Yaskawa INFORM job: DEMO_ROOF_UPPER_0625_3PAINT_39.JBI

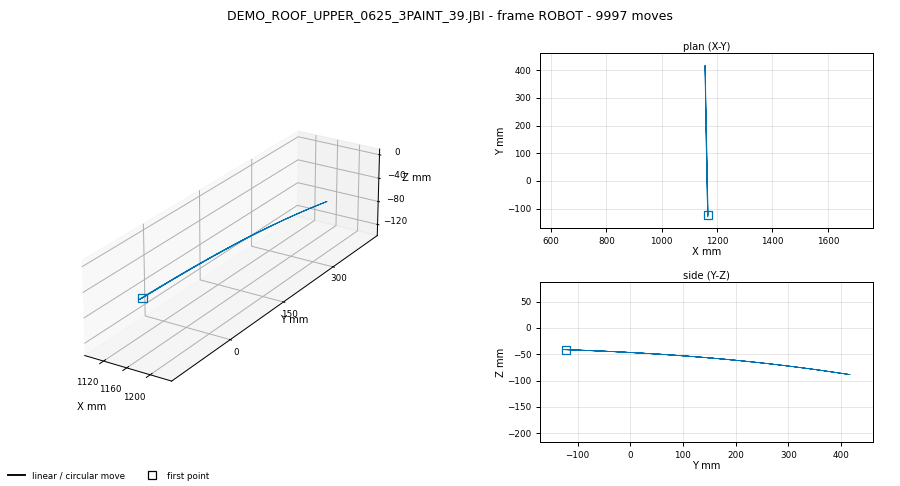
[picture p0: tool path of DEMO_ROOF_UPPER_0625_3PAINT_39.JBI in frame ROBOT, 9997 of 9997 moves have a stored position in this frame; points joined in program order, loops and branches not executed]
/JOB
//NAME DEMO_ROOF_UPPER_0625_3PAINT39
//POS
///NPOS 9997,0,0,0,0,0
///TOOL 0
///USER 0
///POSTYPE ROBOT
///RECTAN
///RCONF 1,0,0,0,0,0,0,0,0,0,0,0,0,0,0,0,0,0,0,0,0,0,0,0
C00000=1167.376,-121.731,-41.179,178.758,5.790,149.399
C00001=1167.371,-121.482,-41.188,178.760,5.791,149.399
C00002=1167.365,-121.231,-41.196,178.762,5.791,149.398
C00003=1167.360,-120.981,-41.205,178.764,5.791,149.397
C00004=1167.355,-120.731,-41.214,178.766,5.791,149.397
C00005=1167.349,-120.482,-41.223,178.768,5.792,149.396
C00006=1167.344,-120.232,-41.232,178.770,5.791,149.396
C00007=1167.339,-119.983,-41.241,178.772,5.792,149.395
C00008=1167.334,-119.733,-41.249,178.774,5.792,149.395
C00009=1167.329,-119.483,-41.258,178.777,5.792,149.394
C00010=1167.323,-119.234,-41.267,178.778,5.792,149.394
C00011=1167.318,-118.984,-41.276,178.780,5.793,149.393
C00012=1167.313,-118.734,-41.285,178.782,5.793,149.393
C00013=1167.307,-118.484,-41.294,178.785,5.793,149.392
C00014=1167.301,-118.233,-41.302,178.786,5.793,149.391
C00015=1167.295,-117.984,-41.311,178.789,5.794,149.391
C00016=1167.290,-117.734,-41.320,178.791,5.794,149.390
C00017=1167.285,-117.485,-41.329,178.793,5.795,149.390
C00018=1167.280,-117.235,-41.338,178.795,5.795,149.389
C00019=1167.275,-116.985,-41.346,178.797,5.795,149.388
C00020=1167.270,-116.735,-41.355,178.799,5.796,149.388
C00021=1167.264,-116.485,-41.364,178.801,5.796,149.387
C00022=1167.259,-116.236,-41.373,178.804,5.796,149.387
C00023=1167.253,-115.986,-41.382,178.805,5.796,149.386
C00024=1167.248,-115.736,-41.391,178.807,5.797,149.386
C00025=1167.242,-115.486,-41.400,178.809,5.796,149.385
C00026=1167.237,-115.236,-41.409,178.812,5.797,149.385
C00027=1167.232,-114.986,-41.418,178.813,5.797,149.384
C00028=1167.226,-114.737,-41.426,178.816,5.797,149.383
C00029=1167.220,-114.487,-41.436,178.817,5.797,149.383
C00030=1167.216,-114.238,-41.446,178.820,5.798,149.382
C00031=1167.210,-113.988,-41.454,178.822,5.798,149.382
C00032=1167.205,-113.738,-41.463,178.824,5.798,149.381
C00033=1167.200,-113.488,-41.472,178.826,5.798,149.381
C00034=1167.195,-113.238,-41.481,178.828,5.799,149.380
C00035=1167.189,-112.988,-41.491,178.830,5.799,149.380
C00036=1167.184,-112.738,-41.500,178.832,5.800,149.379
C00037=1167.178,-112.489,-41.508,178.835,5.800,149.378
C00038=1167.173,-112.239,-41.517,178.836,5.800,149.378
C00039=1167.168,-111.990,-41.526,178.839,5.801,149.377
C00040=1167.162,-111.739,-41.535,178.841,5.800,149.377
C00041=1167.157,-111.490,-41.545,178.843,5.801,149.376
C00042=1167.152,-111.240,-41.554,178.844,5.801,149.376
C00043=1167.147,-110.991,-41.563,178.847,5.801,149.375
C00044=1167.141,-110.741,-41.572,178.849,5.801,149.374
C00045=1167.136,-110.490,-41.581,178.851,5.802,149.374
C00046=1167.130,-110.241,-41.590,178.853,5.802,149.373
C00047=1167.125,-109.991,-41.599,178.855,5.802,149.373
C00048=1167.120,-109.742,-41.608,178.858,5.803,149.372
C00049=1167.114,-109.492,-41.618,178.859,5.803,149.372
C00050=1167.109,-109.242,-41.627,178.862,5.804,149.371
C00051=1167.104,-108.992,-41.635,178.864,5.803,149.370
C00052=1167.098,-108.743,-41.644,178.866,5.804,149.370
C00053=1167.092,-108.492,-41.654,178.867,5.804,149.369
C00054=1167.088,-108.243,-41.663,178.870,5.804,149.369
C00055=1167.082,-107.993,-41.672,178.872,5.804,149.368
C00056=1167.077,-107.743,-41.681,178.874,5.805,149.368
C00057=1167.071,-107.493,-41.691,178.876,5.805,149.367
C00058=1167.067,-107.244,-41.700,178.878,5.805,149.367
C00059=1167.061,-106.994,-41.709,178.881,5.806,149.366
C00060=1167.055,-106.744,-41.719,178.882,5.806,149.365
C00061=1167.050,-106.494,-41.728,178.885,5.806,149.365
C00062=1167.045,-106.245,-41.737,178.887,5.806,149.364
C00063=1167.040,-105.995,-41.747,178.889,5.807,149.364
C00064=1167.034,-105.745,-41.756,178.891,5.807,149.363
C00065=1167.029,-105.495,-41.765,178.893,5.807,149.362
C00066=1167.024,-105.246,-41.775,178.895,5.808,149.362
C00067=1167.018,-104.996,-41.784,178.897,5.808,149.361
C00068=1167.013,-104.746,-41.793,178.900,5.808,149.361
C00069=1167.008,-104.496,-41.803,178.901,5.808,149.360
C00070=1167.002,-104.246,-41.812,178.904,5.809,149.360
C00071=1166.997,-103.997,-41.821,178.906,5.809,149.359
C00072=1166.992,-103.747,-41.831,178.908,5.809,149.359
C00073=1166.987,-103.497,-41.840,178.910,5.809,149.358
C00074=1166.981,-103.247,-41.849,178.912,5.810,149.357
C00075=1166.976,-102.998,-41.859,178.915,5.810,149.357
C00076=1166.971,-102.748,-41.868,178.916,5.810,149.356
C00077=1166.965,-102.476,-41.878,178.919,5.810,149.356
C00078=1166.960,-102.204,-41.888,178.921,5.811,149.355
C00079=1166.953,-101.933,-41.899,178.923,5.811,149.354
C00080=1166.947,-101.661,-41.909,178.925,5.812,149.354
C00081=1166.942,-101.411,-41.918,178.928,5.812,149.353
C00082=1166.937,-101.161,-41.928,178.930,5.812,149.353
C00083=1166.931,-100.911,-41.937,178.932,5.812,149.352
C00084=1166.926,-100.662,-41.946,178.934,5.812,149.351
C00085=1166.921,-100.412,-41.956,178.936,5.813,149.351
C00086=1166.916,-100.161,-41.965,178.939,5.813,149.350
C00087=1166.910,-99.912,-41.975,178.940,5.813,149.350
C00088=1166.905,-99.662,-41.984,178.943,5.814,149.349
C00089=1166.899,-99.412,-41.994,178.945,5.814,149.349
C00090=1166.895,-99.163,-42.003,178.947,5.815,149.348
C00091=1166.889,-98.913,-42.013,178.949,5.814,149.347
C00092=1166.884,-98.663,-42.023,178.951,5.815,149.347
C00093=1166.879,-98.413,-42.031,178.954,5.815,149.346
C00094=1166.873,-98.164,-42.042,178.955,5.815,149.346
C00095=1166.868,-97.914,-42.051,178.958,5.816,149.345
C00096=1166.862,-97.665,-42.061,178.960,5.816,149.344
C00097=1166.857,-97.415,-42.070,178.962,5.816,149.344
C00098=1166.851,-97.165,-42.080,178.965,5.817,149.343
C00099=1166.846,-96.915,-42.089,178.966,5.817,149.343
C00100=1166.841,-96.665,-42.099,178.968,5.818,149.342
C00101=1166.836,-96.415,-42.108,178.970,5.817,149.342
C00102=1166.831,-96.166,-42.118,178.973,5.818,149.341
C00103=1166.825,-95.916,-42.127,178.975,5.818,149.340
C00104=1166.820,-95.666,-42.138,178.977,5.818,149.340
C00105=1166.815,-95.416,-42.146,178.980,5.819,149.339
C00106=1166.809,-95.167,-42.157,178.981,5.819,149.339
C00107=1166.804,-94.918,-42.166,178.983,5.819,149.338
C00108=1166.798,-94.667,-42.176,178.986,5.820,149.338
C00109=1166.793,-94.417,-42.186,178.988,5.820,149.337
C00110=1166.788,-94.167,-42.195,178.990,5.820,149.336
C00111=1166.782,-93.918,-42.205,178.992,5.820,149.336
C00112=1166.777,-93.668,-42.214,178.994,5.821,149.335
C00113=1166.772,-93.418,-42.225,178.997,5.821,149.335
C00114=1166.767,-93.169,-42.234,178.998,5.821,149.334
C00115=1166.761,-92.919,-42.244,179.001,5.822,149.333
C00116=1166.757,-92.669,-42.254,179.003,5.822,149.333
C00117=1166.751,-92.419,-42.263,179.005,5.822,149.332
C00118=1166.745,-92.169,-42.273,179.008,5.823,149.332
C00119=1166.740,-91.920,-42.283,179.009,5.823,149.331
C00120=1166.734,-91.670,-42.292,179.012,5.823,149.331
C00121=1166.730,-91.421,-42.302,179.014,5.824,149.330
C00122=1166.725,-91.170,-42.313,179.016,5.824,149.329
C00123=1166.719,-90.920,-42.322,179.018,5.824,149.329
C00124=1166.714,-90.671,-42.332,179.020,5.824,149.328
C00125=1166.708,-90.422,-42.342,179.023,5.825,149.328
C00126=1166.703,-90.172,-42.351,179.025,5.825,149.327
C00127=1166.698,-89.921,-42.361,179.027,5.825,149.327
C00128=1166.692,-89.672,-42.372,179.029,5.826,149.326
C00129=1166.688,-89.423,-42.381,179.032,5.826,149.325
C00130=1166.682,-89.173,-42.391,179.033,5.826,149.325
C00131=1166.676,-88.923,-42.401,179.036,5.827,149.324
C00132=1166.672,-88.673,-42.411,179.038,5.827,149.324
C00133=1166.666,-88.423,-42.420,179.040,5.827,149.323
C00134=1166.660,-88.173,-42.431,179.042,5.828,149.322
C00135=1166.655,-87.924,-42.440,179.044,5.828,149.322
C00136=1166.650,-87.675,-42.450,179.047,5.828,149.321
C00137=1166.645,-87.424,-42.460,179.049,5.829,149.321
C00138=1166.640,-87.174,-42.470,179.051,5.829,149.320
C00139=1166.634,-86.925,-42.480,179.053,5.829,149.320
C00140=1166.629,-86.675,-42.490,179.056,5.830,149.319
C00141=1166.624,-86.425,-42.500,179.057,5.830,149.318
C00142=1166.618,-86.175,-42.510,179.060,5.830,149.318
C00143=1166.613,-85.926,-42.520,179.062,5.830,149.317
C00144=1166.608,-85.677,-42.530,179.064,5.830,149.316
C00145=1166.603,-85.426,-42.540,179.067,5.831,149.316
C00146=1166.597,-85.177,-42.550,179.068,5.831,149.316
C00147=1166.592,-84.927,-42.560,179.071,5.832,149.315
C00148=1166.587,-84.677,-42.569,179.073,5.832,149.314
C00149=1166.582,-84.427,-42.580,179.075,5.832,149.314
C00150=1166.576,-84.178,-42.590,179.077,5.833,149.313
C00151=1166.571,-83.928,-42.600,179.080,5.833,149.312
C00152=1166.566,-83.678,-42.610,179.082,5.833,149.312
C00153=1166.560,-83.429,-42.621,179.084,5.833,149.311
C00154=1166.555,-83.179,-42.631,179.086,5.834,149.311
C00155=1166.550,-82.929,-42.640,179.088,5.834,149.310
C00156=1166.545,-82.679,-42.650,179.091,5.835,149.310
C00157=1166.539,-82.429,-42.661,179.093,5.835,149.309
C00158=1166.534,-82.180,-42.671,179.095,5.835,149.308
C00159=1166.529,-81.930,-42.681,179.097,5.836,149.308
C00160=1166.524,-81.680,-42.691,179.099,5.835,149.307
C00161=1166.518,-81.431,-42.701,179.101,5.836,149.307
C00162=1166.512,-81.181,-42.711,179.104,5.837,149.306
C00163=1166.507,-80.931,-42.722,179.106,5.837,149.306
C00164=1166.502,-80.681,-42.732,179.108,5.837,149.305
C00165=1166.497,-80.432,-42.742,179.111,5.838,149.304
C00166=1166.492,-80.182,-42.752,179.113,5.837,149.304
C00167=1166.486,-79.932,-42.763,179.115,5.838,149.303
C00168=1166.481,-79.683,-42.773,179.117,5.839,149.302
C00169=1166.476,-79.433,-42.783,179.119,5.839,149.302
C00170=1166.471,-79.183,-42.793,179.122,5.839,149.301
C00171=1166.465,-78.934,-42.803,179.124,5.840,149.301
C00172=1166.460,-78.684,-42.814,179.126,5.839,149.300
C00173=1166.455,-78.434,-42.824,179.128,5.840,149.300
C00174=1166.449,-78.185,-42.834,179.131,5.840,149.299
C00175=1166.444,-77.934,-42.845,179.132,5.840,149.298
C00176=1166.439,-77.685,-42.855,179.135,5.841,149.298
C00177=1166.433,-77.435,-42.865,179.137,5.842,149.297
C00178=1166.429,-77.185,-42.875,179.140,5.842,149.296
C00179=1166.423,-76.936,-42.885,179.142,5.842,149.296
C00180=1166.418,-76.685,-42.896,179.144,5.843,149.295
C00181=1166.412,-76.415,-42.907,179.146,5.843,149.295
C00182=1166.406,-76.143,-42.918,179.149,5.844,149.294
C00183=1166.400,-75.872,-42.930,179.151,5.843,149.293
C00184=1166.395,-75.601,-42.940,179.153,5.844,149.293
C00185=1166.390,-75.351,-42.951,179.156,5.844,149.292
C00186=1166.384,-75.102,-42.962,179.158,5.845,149.292
C00187=1166.379,-74.852,-42.972,179.160,5.845,149.291
C00188=1166.374,-74.602,-42.982,179.162,5.846,149.291
C00189=1166.368,-74.353,-42.993,179.165,5.846,149.290
C00190=1166.363,-74.102,-43.003,179.167,5.846,149.289
C00191=1166.358,-73.853,-43.013,179.169,5.846,149.289
C00192=1166.352,-73.603,-43.024,179.172,5.847,149.288
C00193=1166.347,-73.353,-43.034,179.174,5.847,149.287
C00194=1166.342,-73.104,-43.045,179.176,5.847,149.287
C00195=1166.337,-72.854,-43.056,179.179,5.848,149.286
C00196=1166.331,-72.604,-43.066,179.180,5.848,149.286
C00197=1166.326,-72.355,-43.076,179.183,5.848,149.285
C00198=1166.321,-72.104,-43.087,179.185,5.849,149.285
C00199=1166.315,-71.856,-43.098,179.188,5.849,149.284
C00200=1166.310,-71.605,-43.108,179.189,5.849,149.283
C00201=1166.305,-71.356,-43.118,179.192,5.850,149.283
C00202=1166.300,-71.106,-43.129,179.194,5.851,149.282
C00203=1166.294,-70.856,-43.139,179.196,5.850,149.281
C00204=1166.289,-70.606,-43.150,179.198,5.851,149.281
C00205=1166.284,-70.357,-43.161,179.201,5.851,149.280
C00206=1166.278,-70.107,-43.171,179.203,5.852,149.280
C00207=1166.273,-69.857,-43.181,179.205,5.852,149.279
C00208=1166.268,-69.608,-43.192,179.208,5.853,149.279
C00209=1166.263,-69.358,-43.203,179.210,5.853,149.278
C00210=1166.257,-69.108,-43.213,179.212,5.853,149.277
C00211=1166.252,-68.858,-43.224,179.214,5.853,149.277
C00212=1166.247,-68.609,-43.235,179.217,5.854,149.276
C00213=1166.242,-68.359,-43.245,179.219,5.855,149.276
C00214=1166.236,-68.109,-43.255,179.221,5.855,149.275
C00215=1166.232,-67.860,-43.267,179.224,5.855,149.274
C00216=1166.226,-67.610,-43.277,179.226,5.856,149.274
C00217=1166.220,-67.360,-43.288,179.228,5.855,149.273
C00218=1166.215,-67.111,-43.299,179.230,5.856,149.273
C00219=1166.210,-66.860,-43.310,179.233,5.857,149.272
C00220=1166.204,-66.611,-43.320,179.235,5.857,149.271
C00221=1166.200,-66.361,-43.331,179.237,5.857,149.271
C00222=1166.194,-66.112,-43.341,179.239,5.858,149.270
C00223=1166.189,-65.862,-43.352,179.242,5.858,149.270
C00224=1166.184,-65.613,-43.363,179.243,5.858,149.269
C00225=1166.179,-65.362,-43.373,179.246,5.859,149.268
C00226=1166.173,-65.113,-43.385,179.248,5.859,149.268
C00227=1166.168,-64.863,-43.395,179.251,5.860,149.267
C00228=1166.162,-64.613,-43.406,179.253,5.860,149.267
C00229=1166.158,-64.364,-43.417,179.255,5.860,149.266
C00230=1166.153,-64.113,-43.428,179.257,5.861,149.266
C00231=1166.147,-63.865,-43.438,179.260,5.861,149.265
C00232=1166.142,-63.614,-43.449,179.262,5.861,149.264
C00233=1166.136,-63.365,-43.461,179.264,5.862,149.264
C00234=1166.131,-63.115,-43.471,179.267,5.862,149.263
C00235=1166.126,-62.865,-43.481,179.269,5.863,149.262
C00236=1166.121,-62.616,-43.493,179.271,5.863,149.262
C00237=1166.116,-62.365,-43.503,179.273,5.863,149.261
C00238=1166.111,-62.116,-43.514,179.276,5.864,149.261
C00239=1166.105,-61.866,-43.525,179.278,5.865,149.260
C00240=1166.100,-61.617,-43.536,179.280,5.864,149.259
C00241=1166.095,-61.367,-43.547,179.283,5.865,149.259
C00242=1166.089,-61.118,-43.558,179.285,5.865,149.258
C00243=1166.084,-60.868,-43.568,179.287,5.866,149.258
C00244=1166.079,-60.618,-43.580,179.289,5.866,149.257
C00245=1166.073,-60.368,-43.590,179.292,5.867,149.257
C00246=1166.069,-60.118,-43.602,179.294,5.867,149.256
C00247=1166.063,-59.870,-43.613,179.297,5.868,149.255
C00248=1166.058,-59.619,-43.624,179.299,5.867,149.255
C00249=1166.053,-59.369,-43.635,179.301,5.868,149.254
C00250=1166.047,-59.120,-43.645,179.303,5.869,149.254
C00251=1166.043,-58.870,-43.657,179.306,5.869,149.253
C00252=1166.037,-58.620,-43.668,179.308,5.869,149.252
C00253=1166.032,-58.371,-43.679,179.310,5.869,149.252
C00254=1166.027,-58.121,-43.690,179.313,5.870,149.251
C00255=1166.021,-57.872,-43.700,179.315,5.871,149.250
C00256=1166.016,-57.622,-43.712,179.317,5.871,149.250
C00257=1166.011,-57.371,-43.723,179.320,5.871,149.249
C00258=1166.006,-57.122,-43.734,179.322,5.872,149.249
C00259=1166.001,-56.873,-43.745,179.324,5.872,149.248
C00260=1165.995,-56.622,-43.756,179.327,5.873,149.248
C00261=1165.990,-56.373,-43.767,179.329,5.873,149.247
C00262=1165.985,-56.124,-43.778,179.331,5.873,149.246
C00263=1165.979,-55.873,-43.789,179.333,5.874,149.246
C00264=1165.974,-55.624,-43.800,179.336,5.875,149.245
C00265=1165.969,-55.375,-43.812,179.338,5.874,149.245
C00266=1165.964,-55.124,-43.823,179.340,5.875,149.244
C00267=1165.958,-54.875,-43.834,179.343,5.875,149.243
C00268=1165.954,-54.626,-43.845,179.345,5.876,149.243
C00269=1165.948,-54.375,-43.856,179.347,5.876,149.242
C00270=1165.943,-54.126,-43.867,179.350,5.876,149.241
C00271=1165.938,-53.876,-43.878,179.352,5.877,149.241
C00272=1165.933,-53.626,-43.890,179.354,5.877,149.240
C00273=1165.928,-53.376,-43.901,179.357,5.878,149.240
C00274=1165.922,-53.127,-43.912,179.359,5.878,149.239
C00275=1165.917,-52.877,-43.924,179.361,5.879,149.239
C00276=1165.912,-52.628,-43.935,179.363,5.879,149.238
C00277=1165.906,-52.378,-43.946,179.366,5.880,149.237
C00278=1165.901,-52.128,-43.957,179.368,5.880,149.237
C00279=1165.896,-51.879,-43.968,179.370,5.880,149.236
C00280=1165.891,-51.629,-43.980,179.373,5.881,149.236
C00281=1165.885,-51.379,-43.990,179.375,5.881,149.235
C00282=1165.880,-51.129,-44.002,179.377,5.882,149.234
C00283=1165.875,-50.880,-44.014,179.380,5.882,149.234
C00284=1165.871,-50.630,-44.025,179.382,5.882,149.233
C00285=1165.864,-50.360,-44.037,179.384,5.883,149.232
C00286=1165.859,-50.089,-44.050,179.387,5.883,149.232
C00287=1165.853,-49.819,-44.062,179.390,5.884,149.231
C00288=1165.847,-49.548,-44.074,179.392,5.884,149.231
C00289=1165.842,-49.298,-44.086,179.395,5.885,149.230
C00290=1165.837,-49.049,-44.097,179.397,5.886,149.229
C00291=1165.832,-48.800,-44.108,179.399,5.886,149.229
C00292=1165.826,-48.550,-44.120,179.401,5.886,149.228
C00293=1165.822,-48.300,-44.131,179.404,5.886,149.228
C00294=1165.816,-48.049,-44.142,179.406,5.887,149.227
C00295=1165.811,-47.801,-44.153,179.409,5.888,149.226
C00296=1165.805,-47.551,-44.165,179.411,5.888,149.226
C00297=1165.801,-47.301,-44.176,179.413,5.888,149.225
C00298=1165.795,-47.051,-44.188,179.415,5.888,149.224
C00299=1165.790,-46.801,-44.200,179.418,5.889,149.224
C00300=1165.784,-46.552,-44.211,179.420,5.890,149.223
C00301=1165.779,-46.302,-44.223,179.423,5.890,149.223
C00302=1165.774,-46.053,-44.234,179.425,5.891,149.222
C00303=1165.769,-45.803,-44.246,179.427,5.890,149.221
C00304=1165.764,-45.553,-44.257,179.429,5.891,149.221
C00305=1165.758,-45.304,-44.269,179.432,5.892,149.220
C00306=1165.753,-45.054,-44.280,179.434,5.893,149.220
C00307=1165.748,-44.804,-44.292,179.437,5.893,149.219
C00308=1165.743,-44.555,-44.303,179.439,5.894,149.219
C00309=1165.738,-44.305,-44.315,179.441,5.893,149.218
C00310=1165.733,-44.056,-44.326,179.444,5.894,149.217
C00311=1165.727,-43.806,-44.338,179.446,5.895,149.217
C00312=1165.722,-43.556,-44.350,179.449,5.895,149.216
C00313=1165.717,-43.306,-44.361,179.451,5.896,149.216
C00314=1165.712,-43.056,-44.373,179.454,5.896,149.215
C00315=1165.707,-42.807,-44.384,179.455,5.896,149.214
C00316=1165.702,-42.557,-44.396,179.458,5.897,149.214
C00317=1165.695,-42.308,-44.408,179.460,5.897,149.213
C00318=1165.691,-42.058,-44.419,179.463,5.898,149.212
C00319=1165.685,-41.808,-44.431,179.465,5.898,149.212
C00320=1165.680,-41.558,-44.443,179.467,5.899,149.211
C00321=1165.675,-41.308,-44.454,179.470,5.899,149.211
C00322=1165.670,-41.059,-44.467,179.472,5.900,149.210
C00323=1165.665,-40.809,-44.478,179.474,5.900,149.209
C00324=1165.660,-40.560,-44.490,179.477,5.901,149.209
C00325=1165.654,-40.310,-44.502,179.479,5.901,149.208
C00326=1165.649,-40.061,-44.513,179.482,5.902,149.208
C00327=1165.644,-39.811,-44.525,179.484,5.902,149.207
C00328=1165.638,-39.561,-44.537,179.486,5.902,149.206
C00329=1165.634,-39.312,-44.549,179.488,5.903,149.206
C00330=1165.629,-39.062,-44.560,179.491,5.903,149.205
C00331=1165.623,-38.812,-44.572,179.493,5.904,149.205
C00332=1165.618,-38.562,-44.584,179.496,5.904,149.204
C00333=1165.613,-38.312,-44.596,179.498,5.905,149.204
C00334=1165.607,-38.063,-44.607,179.501,5.906,149.203
C00335=1165.602,-37.814,-44.620,179.503,5.905,149.202
C00336=1165.597,-37.564,-44.631,179.505,5.906,149.202
C00337=1165.592,-37.314,-44.643,179.508,5.907,149.201
C00338=1165.586,-37.064,-44.655,179.510,5.907,149.201
C00339=1165.581,-36.815,-44.667,179.512,5.908,149.200
C00340=1165.577,-36.565,-44.679,179.515,5.909,149.199
C00341=1165.571,-36.315,-44.691,179.517,5.909,149.199
C00342=1165.566,-36.065,-44.702,179.519,5.909,149.198
C00343=1165.561,-35.816,-44.715,179.522,5.909,149.197
C00344=1165.556,-35.567,-44.726,179.524,5.910,149.197
C00345=1165.550,-35.317,-44.738,179.526,5.911,149.196
C00346=1165.545,-35.067,-44.750,179.529,5.911,149.196
C00347=1165.540,-34.817,-44.763,179.531,5.912,149.195
C00348=1165.535,-34.568,-44.774,179.534,5.912,149.194
C00349=1165.530,-34.318,-44.786,179.537,5.913,149.194
C00350=1165.525,-34.068,-44.798,179.539,5.914,149.193
C00351=1165.519,-33.819,-44.810,179.541,5.913,149.193
C00352=1165.514,-33.569,-44.822,179.543,5.914,149.192
C00353=1165.509,-33.320,-44.834,179.546,5.914,149.191
C00354=1165.504,-33.070,-44.846,179.548,5.915,149.191
C00355=1165.499,-32.820,-44.858,179.551,5.916,149.190
C00356=1165.493,-32.570,-44.871,179.553,5.916,149.190
C00357=1165.488,-32.320,-44.882,179.555,5.917,149.189
C00358=1165.483,-32.071,-44.895,179.558,5.917,149.188
C00359=1165.478,-31.822,-44.906,179.560,5.918,149.188
C00360=1165.473,-31.572,-44.918,179.562,5.918,149.187
C00361=1165.468,-31.322,-44.931,179.564,5.919,149.187
C00362=1165.462,-31.072,-44.943,179.567,5.919,149.186
C00363=1165.457,-30.823,-44.955,179.570,5.919,149.185
C00364=1165.452,-30.573,-44.967,179.572,5.920,149.185
C00365=1165.446,-30.323,-44.979,179.575,5.921,149.184
C00366=1165.442,-30.074,-44.991,179.577,5.921,149.184
C00367=1165.436,-29.824,-45.003,179.579,5.922,149.183
C00368=1165.431,-29.575,-45.016,179.582,5.923,149.182
C00369=1165.426,-29.325,-45.027,179.584,5.923,149.182
C00370=1165.421,-29.076,-45.040,179.586,5.923,149.181
C00371=1165.415,-28.826,-45.052,179.589,5.924,149.181
C00372=1165.410,-28.576,-45.065,179.591,5.924,149.180
C00373=1165.405,-28.326,-45.076,179.593,5.925,149.179
C00374=1165.400,-28.077,-45.089,179.596,5.925,149.179
C00375=1165.394,-27.827,-45.101,179.598,5.926,149.178
C00376=1165.389,-27.578,-45.114,179.601,5.927,149.178
C00377=1165.385,-27.328,-45.125,179.604,5.927,149.177
C00378=1165.380,-27.078,-45.138,179.606,5.928,149.176
C00379=1165.374,-26.828,-45.150,179.608,5.928,149.176
C00380=1165.369,-26.579,-45.162,179.611,5.929,149.175
C00381=1165.364,-26.330,-45.175,179.613,5.929,149.175
C00382=1165.359,-26.080,-45.187,179.615,5.929,149.174
C00383=1165.354,-25.830,-45.199,179.618,5.930,149.173
C00384=1165.348,-25.580,-45.211,179.620,5.930,149.173
C00385=1165.343,-25.331,-45.224,179.622,5.931,149.172
C00386=1165.338,-25.081,-45.236,179.625,5.932,149.172
C00387=1165.333,-24.831,-45.249,179.627,5.932,149.171
C00388=1165.328,-24.582,-45.261,179.630,5.933,149.170
C00389=1165.322,-24.312,-45.274,179.633,5.933,149.170
C00390=1165.316,-24.042,-45.288,179.635,5.934,149.169
C00391=1165.311,-23.772,-45.301,179.637,5.934,149.169
C00392=1165.305,-23.503,-45.314,179.640,5.935,149.168
C00393=1165.300,-23.254,-45.327,179.643,5.935,149.167
C00394=1165.295,-23.003,-45.339,179.645,5.936,149.167
C00395=1165.290,-22.753,-45.352,179.648,5.937,149.166
C00396=1165.284,-22.504,-45.365,179.650,5.937,149.165
C00397=1165.279,-22.254,-45.377,179.652,5.938,149.165
C00398=1165.274,-22.005,-45.390,179.655,5.938,149.164
C00399=1165.269,-21.755,-45.402,179.657,5.939,149.164
C00400=1165.263,-21.505,-45.414,179.660,5.940,149.163
C00401=1165.259,-21.255,-45.427,179.662,5.940,149.162
C00402=1165.254,-21.006,-45.440,179.665,5.941,149.162
C00403=1165.249,-20.757,-45.452,179.667,5.941,149.161
C00404=1165.243,-20.507,-45.464,179.670,5.942,149.161
C00405=1165.238,-20.257,-45.477,179.672,5.942,149.160
C00406=1165.233,-20.007,-45.490,179.674,5.943,149.159
C00407=1165.228,-19.758,-45.503,179.677,5.944,149.159
C00408=1165.222,-19.508,-45.515,179.679,5.945,149.158
C00409=1165.217,-19.259,-45.527,179.682,5.945,149.158
C00410=1165.212,-19.009,-45.540,179.684,5.945,149.157
C00411=1165.207,-18.759,-45.553,179.686,5.945,149.156
C00412=1165.202,-18.510,-45.566,179.689,5.946,149.156
C00413=1165.197,-18.260,-45.577,179.691,5.947,149.155
C00414=1165.191,-18.010,-45.591,179.694,5.947,149.155
C00415=1165.186,-17.761,-45.603,179.696,5.948,149.154
C00416=1165.181,-17.511,-45.616,179.698,5.948,149.153
C00417=1165.176,-17.262,-45.629,179.701,5.949,149.153
C00418=1165.171,-17.012,-45.641,179.703,5.950,149.152
C00419=1165.166,-16.763,-45.654,179.706,5.950,149.152
C00420=1165.160,-16.512,-45.667,179.708,5.951,149.151
C00421=1165.155,-16.263,-45.679,179.711,5.951,149.150
C00422=1165.150,-16.013,-45.692,179.713,5.952,149.150
C00423=1165.145,-15.764,-45.705,179.716,5.953,149.149
C00424=1165.141,-15.514,-45.718,179.718,5.953,149.149
C00425=1165.135,-15.265,-45.731,179.720,5.954,149.148
C00426=1165.130,-15.015,-45.743,179.723,5.954,149.147
C00427=1165.124,-14.766,-45.756,179.725,5.955,149.147
C00428=1165.120,-14.516,-45.769,179.728,5.956,149.146
C00429=1165.114,-14.266,-45.782,179.731,5.956,149.145
C00430=1165.109,-14.017,-45.795,179.733,5.957,149.145
C00431=1165.104,-13.767,-45.808,179.735,5.957,149.144
C00432=1165.099,-13.518,-45.820,179.738,5.958,149.144
C00433=1165.093,-13.268,-45.834,179.740,5.959,149.143
C00434=1165.088,-13.019,-45.846,179.743,5.959,149.142
C00435=1165.084,-12.769,-45.859,179.745,5.960,149.142
C00436=1165.079,-12.519,-45.872,179.748,5.960,149.141
C00437=1165.073,-12.270,-45.885,179.750,5.961,149.141
C00438=1165.068,-12.020,-45.898,179.753,5.961,149.140
C00439=1165.063,-11.770,-45.910,179.755,5.962,149.140
C00440=1165.057,-11.521,-45.924,179.757,5.963,149.139
C00441=1165.053,-11.271,-45.937,179.760,5.963,149.138
C00442=1165.048,-11.021,-45.949,179.762,5.964,149.138
C00443=1165.042,-10.772,-45.962,179.765,5.964,149.137
C00444=1165.037,-10.522,-45.975,179.767,5.965,149.137
C00445=1165.032,-10.272,-45.988,179.770,5.966,149.136
C00446=1165.026,-10.023,-46.001,179.772,5.966,149.135
C00447=1165.022,-9.773,-46.014,179.775,5.967,149.135
C00448=1165.017,-9.523,-46.027,179.777,5.967,149.134
C00449=1165.011,-9.274,-46.040,179.779,5.968,149.134
C00450=1165.007,-9.024,-46.054,179.782,5.969,149.133
C00451=1165.001,-8.775,-46.066,179.784,5.970,149.133
C00452=1164.996,-8.525,-46.080,179.787,5.970,149.132
C00453=1164.991,-8.275,-46.092,179.790,5.970,149.131
C00454=1164.986,-8.026,-46.105,179.792,5.971,149.131
C00455=1164.981,-7.776,-46.119,179.794,5.972,149.130
C00456=1164.976,-7.526,-46.131,179.797,5.973,149.130
C00457=1164.970,-7.277,-46.145,179.799,5.973,149.129
C00458=1164.965,-7.027,-46.158,179.801,5.974,149.128
C00459=1164.960,-6.778,-46.171,179.804,5.974,149.128
C00460=1164.955,-6.528,-46.184,179.807,5.975,149.127
C00461=1164.950,-6.279,-46.197,179.809,5.976,149.127
C00462=1164.944,-6.030,-46.211,179.812,5.976,149.126
C00463=1164.940,-5.779,-46.224,179.814,5.977,149.125
C00464=1164.934,-5.530,-46.237,179.816,5.977,149.125
C00465=1164.929,-5.280,-46.250,179.819,5.978,149.124
C00466=1164.925,-5.031,-46.263,179.822,5.979,149.124
C00467=1164.919,-4.781,-46.277,179.824,5.980,149.123
C00468=1164.914,-4.531,-46.289,179.827,5.981,149.122
C00469=1164.908,-4.282,-46.303,179.829,5.981,149.122
C00470=1164.904,-4.032,-46.316,179.831,5.982,149.121
C00471=1164.898,-3.783,-46.329,179.834,5.982,149.121
C00472=1164.894,-3.533,-46.342,179.837,5.983,149.120
C00473=1164.888,-3.284,-46.356,179.839,5.984,149.119
C00474=1164.884,-3.034,-46.369,179.842,5.984,149.119
C00475=1164.878,-2.784,-46.382,179.844,5.985,149.118
C00476=1164.874,-2.535,-46.396,179.846,5.985,149.118
C00477=1164.868,-2.285,-46.409,179.849,5.986,149.117
C00478=1164.863,-2.035,-46.422,179.851,5.987,149.116
C00479=1164.858,-1.786,-46.436,179.854,5.987,149.116
C00480=1164.853,-1.537,-46.449,179.856,5.988,149.115
C00481=1164.847,-1.286,-46.462,179.859,5.988,149.115
C00482=1164.842,-1.037,-46.476,179.861,5.989,149.114
C00483=1164.837,-0.787,-46.489,179.864,5.990,149.113
C00484=1164.832,-0.538,-46.503,179.866,5.990,149.113
C00485=1164.827,-0.288,-46.516,179.869,5.992,149.112
C00486=1164.821,-0.039,-46.529,179.872,5.992,149.112
C00487=1164.817,0.211,-46.543,179.874,5.993,149.111
C00488=1164.811,0.460,-46.556,179.876,5.993,149.110
C00489=1164.806,0.710,-46.570,179.879,5.994,149.110
C00490=1164.801,0.959,-46.583,179.881,5.995,149.109
C00491=1164.796,1.209,-46.597,179.884,5.995,149.109
C00492=1164.791,1.458,-46.610,179.886,5.996,149.108
C00493=1164.786,1.728,-46.625,179.889,5.996,149.107
C00494=1164.780,1.997,-46.640,179.891,5.997,149.107
C00495=1164.774,2.267,-46.654,179.895,5.998,149.106
C00496=1164.768,2.536,-46.669,179.897,5.999,149.106
C00497=1164.764,2.785,-46.682,179.900,5.999,149.105
C00498=1164.759,3.036,-46.696,179.902,6.000,149.104
C00499=1164.754,3.284,-46.709,179.904,6.001,149.104
C00500=1164.749,3.535,-46.723,179.907,6.001,149.103
C00501=1164.743,3.784,-46.737,179.909,6.002,149.103
C00502=1164.739,4.034,-46.750,179.912,6.003,149.102
C00503=1164.733,4.283,-46.764,179.915,6.004,149.101
C00504=1164.728,4.532,-46.778,179.917,6.005,149.101
C00505=1164.722,4.782,-46.791,179.919,6.005,149.100
C00506=1164.718,5.031,-46.805,179.922,6.006,149.100
C00507=1164.713,5.282,-46.818,179.925,6.006,149.099
C00508=1164.707,5.531,-46.832,179.927,6.007,149.098
C00509=1164.703,5.780,-46.846,179.930,6.008,149.098
C00510=1164.697,6.030,-46.859,179.932,6.008,149.097
C00511=1164.692,6.280,-46.874,179.934,6.009,149.097
C00512=1164.688,6.530,-46.886,179.937,6.010,149.096
C00513=1164.682,6.779,-46.900,179.940,6.011,149.095
C00514=1164.677,7.028,-46.915,179.942,6.011,149.095
C00515=1164.672,7.279,-46.928,179.945,6.012,149.094
C00516=1164.667,7.527,-46.942,179.947,6.013,149.094
C00517=1164.662,7.777,-46.956,179.949,6.014,149.093
C00518=1164.656,8.027,-46.969,179.952,6.014,149.092
C00519=1164.651,8.276,-46.983,179.954,6.015,149.092
C00520=1164.647,8.526,-46.997,179.957,6.015,149.091
C00521=1164.642,8.775,-47.011,179.960,6.017,149.091
C00522=1164.636,9.025,-47.024,179.962,6.017,149.090
C00523=1164.631,9.275,-47.039,179.965,6.018,149.089
C00524=1164.626,9.524,-47.053,179.967,6.019,149.089
C00525=1164.622,9.773,-47.066,179.970,6.019,149.088
C00526=1164.616,10.024,-47.080,179.972,6.020,149.088
C00527=1164.611,10.273,-47.094,179.975,6.020,149.087
C00528=1164.606,10.522,-47.108,179.977,6.021,149.087
C00529=1164.601,10.772,-47.122,179.979,6.022,149.086
C00530=1164.595,11.022,-47.136,179.983,6.023,149.085
C00531=1164.591,11.271,-47.149,179.985,6.024,149.085
C00532=1164.586,11.521,-47.163,179.987,6.024,149.084
C00533=1164.580,11.770,-47.177,179.990,6.025,149.084
C00534=1164.575,12.019,-47.192,179.992,6.026,149.083
C00535=1164.570,12.269,-47.206,179.995,6.026,149.082
C00536=1164.565,12.519,-47.219,179.997,6.027,149.082
C00537=1164.560,12.768,-47.233,-180.000,6.028,149.081
C00538=1164.555,13.018,-47.248,-179.997,6.029,149.081
C00539=1164.550,13.268,-47.261,-179.995,6.029,149.080
C00540=1164.545,13.517,-47.275,-179.993,6.030,149.080
C00541=1164.540,13.766,-47.290,-179.990,6.031,149.079
C00542=1164.535,14.016,-47.304,-179.987,6.031,149.078
C00543=1164.529,14.265,-47.318,-179.985,6.032,149.078
C00544=1164.525,14.515,-47.332,-179.982,6.033,149.077
C00545=1164.519,14.765,-47.346,-179.980,6.034,149.077
C00546=1164.514,15.015,-47.360,-179.977,6.035,149.076
C00547=1164.509,15.264,-47.374,-179.975,6.035,149.076
C00548=1164.504,15.513,-47.388,-179.972,6.036,149.075
C00549=1164.499,15.763,-47.402,-179.970,6.037,149.074
C00550=1164.494,16.013,-47.417,-179.967,6.038,149.074
C00551=1164.488,16.262,-47.431,-179.964,6.039,149.073
C00552=1164.483,16.512,-47.445,-179.962,6.039,149.073
C00553=1164.478,16.761,-47.459,-179.959,6.040,149.072
C00554=1164.473,17.011,-47.473,-179.957,6.041,149.071
C00555=1164.469,17.261,-47.488,-179.955,6.041,149.071
C00556=1164.463,17.510,-47.502,-179.952,6.043,149.070
C00557=1164.458,17.759,-47.516,-179.949,6.043,149.070
C00558=1164.453,18.009,-47.530,-179.947,6.044,149.069
C00559=1164.448,18.259,-47.544,-179.944,6.045,149.069
C00560=1164.443,18.508,-47.558,-179.942,6.045,149.068
C00561=1164.438,18.758,-47.573,-179.940,6.046,149.067
C00562=1164.433,19.007,-47.587,-179.936,6.047,149.067
C00563=1164.428,19.256,-47.602,-179.934,6.048,149.066
C00564=1164.423,19.506,-47.616,-179.932,6.048,149.066
C00565=1164.418,19.756,-47.630,-179.929,6.049,149.065
C00566=1164.413,20.005,-47.644,-179.927,6.050,149.064
C00567=1164.408,20.255,-47.659,-179.923,6.051,149.064
C00568=1164.403,20.504,-47.673,-179.921,6.052,149.063
C00569=1164.398,20.754,-47.687,-179.919,6.052,149.063
C00570=1164.393,21.004,-47.701,-179.916,6.053,149.062
C00571=1164.388,21.253,-47.716,-179.914,6.054,149.061
C00572=1164.382,21.502,-47.730,-179.912,6.054,149.061
C00573=1164.378,21.751,-47.745,-179.908,6.056,149.060
C00574=1164.373,22.001,-47.759,-179.906,6.057,149.060
C00575=1164.367,22.251,-47.774,-179.904,6.057,149.059
C00576=1164.362,22.501,-47.788,-179.901,6.058,149.059
C00577=1164.357,22.750,-47.803,-179.899,6.058,149.058
C00578=1164.352,23.000,-47.817,-179.896,6.060,149.057
C00579=1164.347,23.249,-47.831,-179.893,6.060,149.057
C00580=1164.342,23.498,-47.845,-179.891,6.061,149.056
C00581=1164.337,23.748,-47.860,-179.889,6.062,149.056
C00582=1164.331,23.998,-47.875,-179.886,6.062,149.055
C00583=1164.327,24.247,-47.890,-179.883,6.064,149.055
C00584=1164.322,24.497,-47.904,-179.881,6.064,149.054
C00585=1164.317,24.746,-47.919,-179.878,6.065,149.054
C00586=1164.312,24.996,-47.933,-179.876,6.066,149.053
C00587=1164.307,25.246,-47.947,-179.872,6.067,149.052
C00588=1164.301,25.496,-47.962,-179.870,6.068,149.052
C00589=1164.296,25.744,-47.977,-179.868,6.068,149.051
C00590=1164.291,25.994,-47.991,-179.866,6.069,149.051
C00591=1164.286,26.243,-48.006,-179.863,6.070,149.050
C00592=1164.282,26.492,-48.021,-179.860,6.071,149.049
C00593=1164.276,26.742,-48.035,-179.857,6.072,149.049
C00594=1164.271,26.992,-48.050,-179.855,6.073,149.048
C00595=1164.266,27.241,-48.065,-179.853,6.073,149.048
C00596=1164.261,27.491,-48.079,-179.850,6.075,149.047
C00597=1164.255,27.760,-48.095,-179.847,6.075,149.047
C00598=1164.250,28.029,-48.111,-179.845,6.076,149.046
C00599=1164.245,28.298,-48.127,-179.841,6.077,149.045
C00600=1164.239,28.567,-48.143,-179.839,6.078,149.045
C00601=1164.234,28.816,-48.157,-179.837,6.078,149.044
C00602=1164.230,29.066,-48.172,-179.834,6.080,149.044
C00603=1164.224,29.316,-48.187,-179.831,6.080,149.043
C00604=1164.219,29.565,-48.202,-179.829,6.081,149.042
C00605=1164.214,29.814,-48.216,-179.826,6.082,149.042
C00606=1164.209,30.064,-48.232,-179.823,6.083,149.041
C00607=1164.204,30.313,-48.246,-179.821,6.084,149.041
C00608=1164.199,30.563,-48.261,-179.818,6.084,149.040
C00609=1164.194,30.812,-48.275,-179.816,6.085,149.040
C00610=1164.189,31.062,-48.291,-179.813,6.086,149.039
C00611=1164.184,31.311,-48.305,-179.811,6.087,149.038
C00612=1164.179,31.560,-48.320,-179.808,6.088,149.038
C00613=1164.174,31.811,-48.335,-179.806,6.089,149.037
C00614=1164.169,32.060,-48.350,-179.803,6.090,149.037
C00615=1164.163,32.310,-48.365,-179.801,6.091,149.036
C00616=1164.159,32.559,-48.380,-179.798,6.091,149.035
C00617=1164.154,32.808,-48.394,-179.796,6.092,149.035
C00618=1164.148,33.058,-48.410,-179.792,6.093,149.034
C00619=1164.143,33.308,-48.424,-179.790,6.094,149.034
C00620=1164.139,33.557,-48.439,-179.788,6.095,149.033
C00621=1164.133,33.806,-48.455,-179.784,6.096,149.033
C00622=1164.128,34.056,-48.469,-179.782,6.097,149.032
C00623=1164.123,34.305,-48.485,-179.780,6.097,149.031
C00624=1164.118,34.555,-48.499,-179.777,6.098,149.031
C00625=1164.113,34.804,-48.515,-179.774,6.099,149.030
C00626=1164.108,35.053,-48.530,-179.772,6.100,149.030
C00627=1164.103,35.303,-48.544,-179.769,6.101,149.029
C00628=1164.098,35.552,-48.559,-179.767,6.102,149.029
C00629=1164.093,35.802,-48.574,-179.764,6.103,149.028
C00630=1164.088,36.052,-48.590,-179.762,6.104,149.028
C00631=1164.083,36.301,-48.605,-179.759,6.104,149.027
C00632=1164.078,36.551,-48.620,-179.756,6.106,149.026
C00633=1164.073,36.800,-48.635,-179.754,6.106,149.026
C00634=1164.068,37.050,-48.650,-179.752,6.107,149.025
C00635=1164.063,37.299,-48.665,-179.749,6.108,149.025
C00636=1164.058,37.548,-48.681,-179.746,6.109,149.024
C00637=1164.053,37.798,-48.695,-179.744,6.110,149.024
C00638=1164.047,38.047,-48.711,-179.741,6.110,149.023
C00639=1164.043,38.297,-48.726,-179.738,6.112,149.022
C00640=1164.038,38.547,-48.741,-179.736,6.112,149.022
C00641=1164.033,38.796,-48.756,-179.733,6.113,149.021
C00642=1164.027,39.046,-48.771,-179.730,6.115,149.021
C00643=1164.023,39.295,-48.786,-179.728,6.115,149.020
C00644=1164.017,39.544,-48.802,-179.725,6.116,149.019
C00645=1164.013,39.793,-48.817,-179.723,6.117,149.019
C00646=1164.007,40.043,-48.832,-179.720,6.118,149.018
C00647=1164.002,40.294,-48.848,-179.718,6.119,149.018
C00648=1163.998,40.543,-48.863,-179.715,6.119,149.017
C00649=1163.992,40.792,-48.878,-179.712,6.121,149.017
C00650=1163.988,41.041,-48.893,-179.710,6.122,149.016
C00651=1163.982,41.290,-48.909,-179.708,6.122,149.016
C00652=1163.977,41.541,-48.925,-179.704,6.124,149.015
C00653=1163.973,41.790,-48.940,-179.702,6.125,149.015
C00654=1163.967,42.040,-48.955,-179.700,6.125,149.014
C00655=1163.962,42.289,-48.970,-179.697,6.127,149.013
C00656=1163.957,42.538,-48.985,-179.694,6.127,149.013
C00657=1163.952,42.788,-49.001,-179.692,6.128,149.012
C00658=1163.948,43.037,-49.016,-179.689,6.129,149.012
C00659=1163.942,43.287,-49.032,-179.687,6.130,149.011
C00660=1163.937,43.536,-49.047,-179.684,6.131,149.011
C00661=1163.932,43.785,-49.062,-179.681,6.132,149.010
C00662=1163.927,44.035,-49.078,-179.679,6.133,149.009
C00663=1163.922,44.285,-49.094,-179.677,6.134,149.009
C00664=1163.917,44.534,-49.109,-179.673,6.135,149.008
C00665=1163.912,44.783,-49.125,-179.671,6.136,149.008
C00666=1163.907,45.033,-49.140,-179.668,6.136,149.007
C00667=1163.903,45.282,-49.155,-179.666,6.138,149.007
C00668=1163.897,45.532,-49.171,-179.663,6.139,149.006
C00669=1163.892,45.781,-49.187,-179.661,6.139,149.006
C00670=1163.888,46.031,-49.202,-179.658,6.141,149.005
C00671=1163.882,46.280,-49.218,-179.656,6.142,149.005
C00672=1163.877,46.530,-49.233,-179.653,6.142,149.004
C00673=1163.872,46.779,-49.249,-179.650,6.144,149.003
C00674=1163.868,47.029,-49.264,-179.648,6.144,149.003
C00675=1163.862,47.278,-49.280,-179.645,6.145,149.002
C00676=1163.857,47.527,-49.296,-179.642,6.146,149.002
C00677=1163.852,47.777,-49.312,-179.640,6.147,149.001
C00678=1163.848,48.026,-49.327,-179.637,6.148,149.001
C00679=1163.842,48.276,-49.343,-179.635,6.149,149.000
C00680=1163.837,48.525,-49.358,-179.632,6.150,148.999
C00681=1163.832,48.775,-49.374,-179.629,6.152,148.999
C00682=1163.827,49.024,-49.389,-179.627,6.152,148.998
C00683=1163.822,49.273,-49.405,-179.624,6.153,148.998
C00684=1163.818,49.523,-49.421,-179.621,6.154,148.997
C00685=1163.812,49.773,-49.437,-179.619,6.155,148.997
C00686=1163.807,50.022,-49.453,-179.616,6.156,148.996
C00687=1163.803,50.272,-49.468,-179.614,6.157,148.996
C00688=1163.798,50.521,-49.484,-179.611,6.158,148.995
C00689=1163.792,50.770,-49.500,-179.608,6.159,148.995
C00690=1163.787,51.020,-49.516,-179.606,6.160,148.994
C00691=1163.782,51.270,-49.531,-179.603,6.161,148.993
C00692=1163.777,51.519,-49.547,-179.600,6.162,148.993
C00693=1163.772,51.769,-49.564,-179.598,6.163,148.992
C00694=1163.768,52.018,-49.579,-179.595,6.163,148.992
C00695=1163.762,52.267,-49.594,-179.593,6.165,148.991
C00696=1163.758,52.517,-49.611,-179.590,6.166,148.991
C00697=1163.752,52.766,-49.626,-179.587,6.167,148.990
C00698=1163.748,53.016,-49.642,-179.585,6.168,148.989
C00699=1163.742,53.265,-49.658,-179.583,6.169,148.989
C00700=1163.737,53.514,-49.674,-179.580,6.170,148.989
C00701=1163.732,53.783,-49.692,-179.577,6.171,148.988
C00702=1163.727,54.052,-49.709,-179.574,6.172,148.987
C00703=1163.721,54.320,-49.726,-179.572,6.173,148.987
C00704=1163.715,54.589,-49.743,-179.569,6.174,148.986
C00705=1163.711,54.838,-49.759,-179.566,6.175,148.985
C00706=1163.706,55.088,-49.775,-179.563,6.176,148.985
C00707=1163.700,55.337,-49.791,-179.561,6.177,148.984
C00708=1163.696,55.587,-49.807,-179.558,6.179,148.984
C00709=1163.691,55.836,-49.822,-179.556,6.179,148.983
C00710=1163.687,56.085,-49.839,-179.552,6.181,148.983
C00711=1163.681,56.335,-49.854,-179.550,6.182,148.982
C00712=1163.676,56.585,-49.870,-179.548,6.182,148.982
C00713=1163.671,56.833,-49.887,-179.545,6.184,148.981
C00714=1163.666,57.083,-49.902,-179.542,6.184,148.981
C00715=1163.661,57.332,-49.919,-179.540,6.186,148.980
C00716=1163.656,57.582,-49.935,-179.537,6.186,148.979
C00717=1163.651,57.832,-49.952,-179.535,6.187,148.979
C00718=1163.645,58.081,-49.967,-179.531,6.189,148.978
C00719=1163.641,58.330,-49.984,-179.529,6.189,148.978
C00720=1163.636,58.580,-50.000,-179.526,6.191,148.977
C00721=1163.631,58.829,-50.016,-179.524,6.192,148.977
C00722=1163.626,59.079,-50.032,-179.521,6.193,148.976
C00723=1163.621,59.328,-50.049,-179.519,6.194,148.976
C00724=1163.616,59.578,-50.064,-179.516,6.195,148.975
C00725=1163.611,59.827,-50.081,-179.513,6.196,148.975
C00726=1163.606,60.076,-50.097,-179.511,6.197,148.974
C00727=1163.602,60.326,-50.113,-179.508,6.198,148.974
C00728=1163.596,60.575,-50.129,-179.506,6.199,148.973
C00729=1163.592,60.825,-50.145,-179.502,6.200,148.972
C00730=1163.587,61.074,-50.162,-179.500,6.201,148.972
C00731=1163.581,61.323,-50.179,-179.497,6.202,148.971
C00732=1163.576,61.573,-50.195,-179.495,6.203,148.971
C00733=1163.571,61.822,-50.211,-179.492,6.204,148.970
C00734=1163.566,62.071,-50.227,-179.490,6.206,148.970
C00735=1163.562,62.321,-50.243,-179.487,6.206,148.969
C00736=1163.557,62.570,-50.260,-179.484,6.208,148.969
C00737=1163.552,62.819,-50.276,-179.482,6.209,148.968
C00738=1163.547,63.070,-50.292,-179.479,6.210,148.968
C00739=1163.541,63.319,-50.309,-179.477,6.211,148.967
C00740=1163.537,63.568,-50.326,-179.473,6.212,148.967
C00741=1163.532,63.818,-50.342,-179.471,6.213,148.966
C00742=1163.527,64.067,-50.358,-179.468,6.214,148.965
C00743=1163.522,64.316,-50.374,-179.466,6.215,148.965
C00744=1163.517,64.566,-50.392,-179.464,6.216,148.965
C00745=1163.512,64.816,-50.408,-179.461,6.217,148.964
C00746=1163.507,65.065,-50.424,-179.458,6.218,148.963
C00747=1163.502,65.314,-50.441,-179.455,6.219,148.963
C00748=1163.497,65.563,-50.457,-179.453,6.220,148.962
C00749=1163.492,65.813,-50.474,-179.450,6.222,148.962
C00750=1163.487,66.063,-50.490,-179.448,6.223,148.961
C00751=1163.482,66.311,-50.507,-179.445,6.224,148.961
C00752=1163.478,66.561,-50.523,-179.442,6.225,148.960
C00753=1163.472,66.810,-50.540,-179.440,6.226,148.960
C00754=1163.468,67.060,-50.557,-179.437,6.227,148.959
C00755=1163.463,67.310,-50.573,-179.434,6.229,148.959
C00756=1163.458,67.558,-50.589,-179.432,6.229,148.958
C00757=1163.452,67.808,-50.606,-179.429,6.231,148.958
C00758=1163.448,68.058,-50.623,-179.427,6.232,148.957
C00759=1163.443,68.306,-50.639,-179.423,6.233,148.956
C00760=1163.438,68.556,-50.656,-179.421,6.234,148.956
C00761=1163.433,68.806,-50.673,-179.418,6.235,148.955
C00762=1163.428,69.055,-50.689,-179.416,6.236,148.955
C00763=1163.423,69.304,-50.707,-179.413,6.237,148.954
C00764=1163.418,69.554,-50.723,-179.411,6.238,148.954
C00765=1163.413,69.803,-50.739,-179.408,6.240,148.953
C00766=1163.408,70.053,-50.756,-179.405,6.240,148.953
C00767=1163.403,70.303,-50.773,-179.402,6.242,148.952
C00768=1163.398,70.551,-50.789,-179.400,6.243,148.952
C00769=1163.393,70.801,-50.806,-179.397,6.244,148.951
C00770=1163.389,71.051,-50.823,-179.394,6.245,148.951
C00771=1163.383,71.299,-50.839,-179.392,6.246,148.950
C00772=1163.378,71.549,-50.857,-179.390,6.247,148.950
C00773=1163.374,71.799,-50.873,-179.386,6.249,148.949
C00774=1163.368,72.048,-50.890,-179.384,6.250,148.949
C00775=1163.363,72.297,-50.907,-179.381,6.251,148.948
C00776=1163.359,72.546,-50.924,-179.379,6.252,148.948
C00777=1163.354,72.796,-50.942,-179.376,6.253,148.947
C00778=1163.349,73.045,-50.958,-179.373,6.254,148.946
C00779=1163.344,73.294,-50.975,-179.371,6.256,148.946
C00780=1163.339,73.544,-50.992,-179.368,6.256,148.945
C00781=1163.334,73.794,-51.009,-179.365,6.258,148.945
C00782=1163.329,74.042,-51.025,-179.363,6.259,148.945
C00783=1163.325,74.292,-51.042,-179.360,6.260,148.944
C00784=1163.319,74.542,-51.059,-179.358,6.261,148.943
C00785=1163.315,74.791,-51.076,-179.355,6.262,148.943
C00786=1163.309,75.040,-51.094,-179.352,6.264,148.942
C00787=1163.305,75.289,-51.110,-179.350,6.265,148.942
C00788=1163.300,75.539,-51.128,-179.347,6.266,148.941
C00789=1163.295,75.789,-51.144,-179.344,6.267,148.941
C00790=1163.289,76.038,-51.161,-179.341,6.268,148.940
C00791=1163.285,76.286,-51.179,-179.339,6.269,148.940
C00792=1163.280,76.536,-51.196,-179.336,6.271,148.939
C00793=1163.275,76.786,-51.212,-179.334,6.271,148.939
C00794=1163.270,77.036,-51.230,-179.331,6.273,148.938
C00795=1163.264,77.285,-51.247,-179.328,6.274,148.938
C00796=1163.260,77.533,-51.264,-179.326,6.275,148.937
C00797=1163.255,77.783,-51.281,-179.323,6.277,148.937
C00798=1163.251,78.033,-51.298,-179.320,6.277,148.936
C00799=1163.246,78.282,-51.316,-179.317,6.279,148.936
C00800=1163.241,78.531,-51.332,-179.315,6.280,148.935
C00801=1163.235,78.781,-51.349,-179.312,6.281,148.935
C00802=1163.230,79.030,-51.367,-179.310,6.282,148.934
C00803=1163.226,79.279,-51.384,-179.307,6.284,148.933
C00804=1163.221,79.529,-51.401,-179.305,6.284,148.933
C00805=1163.215,79.797,-51.419,-179.301,6.286,148.932
C00806=1163.210,80.066,-51.438,-179.299,6.287,148.932
C00807=1163.205,80.334,-51.457,-179.295,6.289,148.931
C00808=1163.199,80.602,-51.476,-179.293,6.290,148.931
C00809=1163.195,80.852,-51.492,-179.290,6.291,148.930
C00810=1163.190,81.101,-51.510,-179.287,6.293,148.930
C00811=1163.185,81.350,-51.527,-179.285,6.294,148.929
C00812=1163.180,81.599,-51.545,-179.282,6.295,148.929
C00813=1163.175,81.849,-51.562,-179.280,6.296,148.928
C00814=1163.170,82.099,-51.579,-179.277,6.297,148.928
C00815=1163.166,82.348,-51.597,-179.274,6.299,148.927
C00816=1163.160,82.598,-51.614,-179.272,6.300,148.927
C00817=1163.155,82.846,-51.632,-179.269,6.301,148.926
C00818=1163.150,83.096,-51.648,-179.266,6.302,148.926
C00819=1163.145,83.345,-51.666,-179.264,6.304,148.925
C00820=1163.140,83.595,-51.684,-179.260,6.305,148.925
C00821=1163.136,83.843,-51.701,-179.258,6.306,148.924
C00822=1163.131,84.093,-51.718,-179.255,6.307,148.924
C00823=1163.126,84.342,-51.736,-179.253,6.308,148.923
C00824=1163.121,84.592,-51.753,-179.250,6.310,148.923
C00825=1163.117,84.841,-51.771,-179.247,6.311,148.922
C00826=1163.111,85.091,-51.788,-179.245,6.312,148.922
C00827=1163.106,85.340,-51.806,-179.242,6.314,148.921
C00828=1163.101,85.590,-51.823,-179.240,6.314,148.921
C00829=1163.097,85.839,-51.841,-179.237,6.316,148.920
C00830=1163.092,86.088,-51.859,-179.234,6.317,148.920
C00831=1163.087,86.338,-51.876,-179.231,6.318,148.919
C00832=1163.082,86.587,-51.894,-179.229,6.320,148.919
C00833=1163.077,86.836,-51.912,-179.227,6.321,148.918
C00834=1163.073,87.086,-51.929,-179.223,6.322,148.918
C00835=1163.067,87.334,-51.946,-179.221,6.324,148.917
C00836=1163.062,87.584,-51.963,-179.219,6.324,148.917
C00837=1163.057,87.833,-51.981,-179.215,6.326,148.916
C00838=1163.052,88.082,-51.999,-179.213,6.327,148.916
C00839=1163.047,88.332,-52.017,-179.210,6.328,148.915
C00840=1163.043,88.581,-52.034,-179.207,6.330,148.915
C00841=1163.038,88.830,-52.052,-179.205,6.331,148.914
C00842=1163.033,89.080,-52.070,-179.202,6.332,148.914
C00843=1163.028,89.330,-52.088,-179.199,6.334,148.913
C00844=1163.023,89.579,-52.106,-179.197,6.335,148.913
C00845=1163.018,89.828,-52.124,-179.194,6.336,148.912
C00846=1163.013,90.078,-52.141,-179.191,6.338,148.912
C00847=1163.008,90.327,-52.159,-179.189,6.338,148.911
C00848=1163.003,90.576,-52.177,-179.186,6.340,148.911
C00849=1162.999,90.825,-52.194,-179.183,6.341,148.910
C00850=1162.994,91.074,-52.212,-179.181,6.342,148.910
C00851=1162.989,91.324,-52.230,-179.178,6.344,148.909
C00852=1162.984,91.573,-52.247,-179.175,6.345,148.909
C00853=1162.979,91.822,-52.265,-179.173,6.346,148.908
C00854=1162.974,92.072,-52.283,-179.170,6.348,148.908
C00855=1162.969,92.321,-52.301,-179.167,6.348,148.907
C00856=1162.964,92.570,-52.319,-179.165,6.350,148.907
C00857=1162.959,92.820,-52.337,-179.162,6.352,148.906
C00858=1162.954,93.069,-52.355,-179.159,6.352,148.906
C00859=1162.949,93.318,-52.373,-179.157,6.354,148.905
C00860=1162.945,93.568,-52.391,-179.154,6.356,148.905
C00861=1162.940,93.817,-52.409,-179.151,6.356,148.904
C00862=1162.935,94.066,-52.427,-179.149,6.358,148.904
C00863=1162.930,94.315,-52.445,-179.146,6.360,148.903
C00864=1162.925,94.565,-52.463,-179.143,6.360,148.903
C00865=1162.921,94.814,-52.481,-179.140,6.362,148.902
C00866=1162.916,95.063,-52.499,-179.138,6.364,148.902
C00867=1162.911,95.312,-52.517,-179.135,6.364,148.901
C00868=1162.906,95.562,-52.535,-179.132,6.366,148.901
C00869=1162.902,95.811,-52.553,-179.130,6.368,148.900
C00870=1162.897,96.060,-52.571,-179.127,6.368,148.900
C00871=1162.892,96.310,-52.589,-179.124,6.370,148.899
C00872=1162.887,96.559,-52.607,-179.122,6.372,148.899
C00873=1162.881,96.808,-52.626,-179.119,6.372,148.899
C00874=1162.876,97.057,-52.644,-179.116,6.374,148.898
C00875=1162.872,97.307,-52.662,-179.114,6.375,148.897
C00876=1162.867,97.556,-52.680,-179.111,6.377,148.897
C00877=1162.862,97.806,-52.698,-179.108,6.378,148.896
C00878=1162.857,98.055,-52.716,-179.105,6.379,148.896
C00879=1162.852,98.304,-52.734,-179.103,6.381,148.896
C00880=1162.847,98.553,-52.752,-179.100,6.382,148.895
C00881=1162.843,98.803,-52.770,-179.097,6.383,148.895
C00882=1162.837,99.053,-52.789,-179.095,6.385,148.894
C00883=1162.832,99.302,-52.807,-179.093,6.386,148.894
C00884=1162.828,99.550,-52.825,-179.089,6.387,148.893
C00885=1162.823,99.799,-52.843,-179.087,6.389,148.893
C00886=1162.819,100.049,-52.862,-179.084,6.391,148.892
C00887=1162.814,100.298,-52.880,-179.081,6.391,148.892
C00888=1162.808,100.548,-52.898,-179.079,6.393,148.891
C00889=1162.803,100.797,-52.916,-179.076,6.395,148.891
C00890=1162.799,101.046,-52.935,-179.074,6.395,148.890
C00891=1162.794,101.296,-52.953,-179.070,6.397,148.890
C00892=1162.789,101.545,-52.971,-179.068,6.399,148.889
C00893=1162.784,101.794,-52.990,-179.065,6.400,148.889
C00894=1162.780,102.043,-53.009,-179.062,6.401,148.888
C00895=1162.775,102.293,-53.027,-179.060,6.402,148.888
C00896=1162.770,102.542,-53.045,-179.057,6.404,148.887
C00897=1162.764,102.791,-53.064,-179.055,6.405,148.887
C00898=1162.760,103.041,-53.083,-179.052,6.406,148.886
C00899=1162.755,103.290,-53.101,-179.049,6.408,148.886
C00900=1162.750,103.539,-53.119,-179.046,6.410,148.886
C00901=1162.745,103.788,-53.137,-179.044,6.411,148.885
C00902=1162.741,104.038,-53.156,-179.041,6.412,148.884
C00903=1162.736,104.287,-53.174,-179.038,6.414,148.884
C00904=1162.730,104.536,-53.193,-179.035,6.415,148.884
C00905=1162.726,104.786,-53.212,-179.033,6.416,148.883
C00906=1162.721,105.035,-53.230,-179.030,6.418,148.883
C00907=1162.716,105.284,-53.249,-179.027,6.419,148.882
C00908=1162.712,105.534,-53.267,-179.025,6.421,148.882
C00909=1162.707,105.802,-53.287,-179.021,6.422,148.881
C00910=1162.701,106.070,-53.308,-179.019,6.423,148.881
C00911=1162.695,106.338,-53.328,-179.016,6.425,148.880
C00912=1162.691,106.607,-53.347,-179.013,6.426,148.880
C00913=1162.686,106.856,-53.366,-179.011,6.428,148.879
C00914=1162.680,107.105,-53.385,-179.008,6.430,148.879
C00915=1162.676,107.355,-53.404,-179.005,6.431,148.878
C00916=1162.671,107.604,-53.422,-179.003,6.432,148.878
C00917=1162.666,107.853,-53.441,-179.000,6.434,148.877
C00918=1162.662,108.102,-53.459,-178.997,6.436,148.877
C00919=1162.657,108.351,-53.479,-178.994,6.437,148.876
C00920=1162.652,108.600,-53.497,-178.992,6.438,148.876
C00921=1162.647,108.850,-53.516,-178.989,6.439,148.876
C00922=1162.642,109.099,-53.534,-178.986,6.441,148.875
C00923=1162.638,109.349,-53.553,-178.983,6.443,148.875
C00924=1162.632,109.598,-53.572,-178.980,6.444,148.874
C00925=1162.628,109.847,-53.591,-178.978,6.445,148.874
C00926=1162.623,110.097,-53.609,-178.976,6.447,148.873
C00927=1162.618,110.345,-53.628,-178.972,6.448,148.873
C00928=1162.613,110.595,-53.648,-178.970,6.450,148.872
C00929=1162.608,110.844,-53.666,-178.968,6.451,148.872
C00930=1162.603,111.093,-53.685,-178.965,6.453,148.871
C00931=1162.599,111.343,-53.703,-178.962,6.454,148.871
C00932=1162.593,111.592,-53.723,-178.959,6.456,148.870
C00933=1162.589,111.841,-53.742,-178.956,6.457,148.870
C00934=1162.584,112.090,-53.760,-178.954,6.458,148.870
C00935=1162.580,112.340,-53.779,-178.951,6.460,148.869
C00936=1162.574,112.589,-53.799,-178.948,6.461,148.869
C00937=1162.570,112.838,-53.817,-178.945,6.463,148.868
C00938=1162.565,113.087,-53.836,-178.943,6.465,148.868
C00939=1162.559,113.336,-53.856,-178.941,6.466,148.867
C00940=1162.555,113.586,-53.874,-178.938,6.467,148.867
C00941=1162.550,113.835,-53.893,-178.935,6.469,148.866
C00942=1162.546,114.084,-53.912,-178.932,6.470,148.866
C00943=1162.540,114.333,-53.932,-178.929,6.472,148.865
C00944=1162.536,114.583,-53.950,-178.927,6.473,148.865
C00945=1162.531,114.832,-53.969,-178.924,6.475,148.865
C00946=1162.526,115.081,-53.989,-178.921,6.476,148.864
C00947=1162.521,115.330,-54.008,-178.918,6.478,148.864
C00948=1162.517,115.579,-54.027,-178.916,6.479,148.863
C00949=1162.511,115.829,-54.046,-178.913,6.481,148.863
C00950=1162.507,116.078,-54.065,-178.911,6.482,148.862
C00951=1162.502,116.327,-54.084,-178.908,6.483,148.862
C00952=1162.497,116.577,-54.104,-178.905,6.485,148.861
C00953=1162.492,116.825,-54.123,-178.902,6.487,148.861
C00954=1162.488,117.075,-54.142,-178.900,6.489,148.861
C00955=1162.482,117.324,-54.161,-178.897,6.490,148.860
C00956=1162.478,117.573,-54.180,-178.894,6.491,148.860
C00957=1162.473,117.822,-54.199,-178.892,6.493,148.859
C00958=1162.468,118.072,-54.219,-178.889,6.494,148.859
C00959=1162.464,118.321,-54.238,-178.886,6.496,148.858
C00960=1162.458,118.570,-54.257,-178.883,6.498,148.858
C00961=1162.454,118.820,-54.277,-178.881,6.498,148.857
C00962=1162.449,119.068,-54.295,-178.878,6.500,148.857
C00963=1162.444,119.318,-54.315,-178.875,6.502,148.857
C00964=1162.439,119.567,-54.334,-178.873,6.503,148.856
C00965=1162.434,119.816,-54.354,-178.870,6.505,148.856
C00966=1162.430,120.065,-54.373,-178.867,6.507,148.855
C00967=1162.425,120.314,-54.392,-178.864,6.508,148.855
C00968=1162.420,120.564,-54.412,-178.862,6.509,148.854
C00969=1162.415,120.813,-54.431,-178.859,6.511,148.854
C00970=1162.410,121.062,-54.451,-178.856,6.513,148.853
C00971=1162.406,121.312,-54.470,-178.854,6.514,148.853
C00972=1162.401,121.560,-54.489,-178.851,6.516,148.853
C00973=1162.396,121.810,-54.509,-178.848,6.517,148.852
C00974=1162.391,122.059,-54.528,-178.845,6.519,148.852
C00975=1162.386,122.308,-54.548,-178.843,6.520,148.851
C00976=1162.382,122.557,-54.568,-178.840,6.522,148.851
C00977=1162.377,122.806,-54.587,-178.838,6.523,148.850
C00978=1162.372,123.055,-54.607,-178.835,6.525,148.850
C00979=1162.367,123.305,-54.626,-178.832,6.526,148.849
C00980=1162.362,123.554,-54.646,-178.829,6.528,148.849
C00981=1162.357,123.804,-54.665,-178.826,6.530,148.849
C00982=1162.353,124.053,-54.684,-178.824,6.532,148.848
C00983=1162.348,124.301,-54.704,-178.821,6.533,148.848
C00984=1162.344,124.551,-54.724,-178.819,6.534,148.847
C00985=1162.339,124.800,-54.744,-178.816,6.536,148.847
C00986=1162.333,125.049,-54.763,-178.813,6.537,148.846
C00987=1162.329,125.299,-54.783,-178.810,6.539,148.846
C00988=1162.324,125.548,-54.803,-178.807,6.541,148.846
C00989=1162.319,125.796,-54.822,-178.805,6.543,148.845
C00990=1162.314,126.046,-54.842,-178.802,6.544,148.845
C00991=1162.309,126.296,-54.862,-178.799,6.546,148.844
C00992=1162.306,126.544,-54.881,-178.797,6.547,148.844
C00993=1162.300,126.793,-54.901,-178.794,6.548,148.843
C00994=1162.296,127.043,-54.920,-178.791,6.550,148.843
C00995=1162.291,127.292,-54.941,-178.789,6.552,148.843
C00996=1162.286,127.541,-54.960,-178.786,6.553,148.842
C00997=1162.281,127.790,-54.980,-178.783,6.555,148.842
C00998=1162.277,128.039,-55.000,-178.780,6.557,148.841
C00999=1162.272,128.289,-55.020,-178.778,6.559,148.841
C01000=1162.267,128.538,-55.039,-178.774,6.560,148.840
C01001=1162.262,128.786,-55.059,-178.772,6.562,148.840
C01002=1162.257,129.036,-55.079,-178.770,6.563,148.840
C01003=1162.253,129.285,-55.099,-178.767,6.564,148.839
C01004=1162.248,129.534,-55.119,-178.764,6.566,148.839
C01005=1162.243,129.783,-55.138,-178.762,6.568,148.838
C01006=1162.238,130.032,-55.159,-178.759,6.569,148.838
C01007=1162.234,130.282,-55.178,-178.756,6.571,148.838
C01008=1162.229,130.531,-55.199,-178.753,6.573,148.837
C01009=1162.223,130.780,-55.219,-178.750,6.574,148.837
C01010=1162.219,131.029,-55.239,-178.747,6.576,148.836
C01011=1162.214,131.278,-55.259,-178.745,6.578,148.836
C01012=1162.210,131.527,-55.279,-178.742,6.579,148.835
C01013=1162.205,131.796,-55.300,-178.739,6.581,148.835
C01014=1162.199,132.065,-55.322,-178.737,6.583,148.835
C01015=1162.194,132.333,-55.344,-178.733,6.584,148.834
C01016=1162.189,132.602,-55.365,-178.731,6.586,148.834
C01017=1162.184,132.852,-55.385,-178.728,6.588,148.833
C01018=1162.179,133.100,-55.405,-178.725,6.589,148.833
C01019=1162.175,133.349,-55.425,-178.723,6.591,148.832
C01020=1162.170,133.598,-55.445,-178.720,6.593,148.832
C01021=1162.165,133.847,-55.465,-178.717,6.595,148.832
C01022=1162.160,134.097,-55.486,-178.714,6.596,148.831
C01023=1162.155,134.346,-55.506,-178.711,6.598,148.831
C01024=1162.151,134.595,-55.526,-178.709,6.599,148.830
C01025=1162.146,134.844,-55.546,-178.706,6.601,148.830
C01026=1162.141,135.093,-55.566,-178.703,6.603,148.830
C01027=1162.136,135.342,-55.587,-178.700,6.605,148.829
C01028=1162.131,135.592,-55.607,-178.698,6.606,148.829
C01029=1162.127,135.841,-55.627,-178.695,6.608,148.828
C01030=1162.122,136.090,-55.647,-178.692,6.610,148.828
C01031=1162.118,136.339,-55.667,-178.690,6.612,148.828
C01032=1162.112,136.588,-55.688,-178.687,6.613,148.827
C01033=1162.108,136.837,-55.708,-178.684,6.615,148.827
C01034=1162.103,137.086,-55.728,-178.682,6.617,148.826
C01035=1162.098,137.335,-55.748,-178.678,6.618,148.826
C01036=1162.093,137.584,-55.769,-178.676,6.619,148.825
C01037=1162.089,137.833,-55.789,-178.674,6.621,148.825
C01038=1162.084,138.082,-55.810,-178.671,6.622,148.825
C01039=1162.079,138.332,-55.830,-178.668,6.624,148.824
C01040=1162.074,138.581,-55.850,-178.665,6.626,148.824
C01041=1162.070,138.830,-55.871,-178.663,6.628,148.823
C01042=1162.065,139.079,-55.891,-178.660,6.629,148.823
C01043=1162.060,139.328,-55.912,-178.657,6.631,148.823
C01044=1162.056,139.577,-55.932,-178.655,6.633,148.822
C01045=1162.051,139.827,-55.952,-178.652,6.635,148.822
C01046=1162.046,140.076,-55.973,-178.649,6.636,148.821
C01047=1162.041,140.325,-55.993,-178.646,6.638,148.821
C01048=1162.036,140.574,-56.014,-178.644,6.640,148.821
C01049=1162.032,140.823,-56.035,-178.641,6.642,148.820
C01050=1162.027,141.072,-56.055,-178.638,6.643,148.820
C01051=1162.022,141.321,-56.076,-178.636,6.645,148.820
C01052=1162.018,141.570,-56.096,-178.633,6.647,148.819
C01053=1162.013,141.819,-56.117,-178.630,6.648,148.819
C01054=1162.008,142.069,-56.138,-178.628,6.650,148.818
C01055=1162.004,142.318,-56.158,-178.624,6.652,148.818
C01056=1161.999,142.567,-56.179,-178.622,6.653,148.817
C01057=1161.994,142.816,-56.200,-178.619,6.655,148.817
C01058=1161.990,143.065,-56.220,-178.616,6.657,148.817
C01059=1161.985,143.314,-56.241,-178.614,6.658,148.816
C01060=1161.980,143.563,-56.261,-178.611,6.660,148.816
C01061=1161.975,143.812,-56.282,-178.608,6.662,148.815
C01062=1161.970,144.061,-56.303,-178.605,6.664,148.815
C01063=1161.965,144.310,-56.324,-178.603,6.665,148.815
C01064=1161.961,144.559,-56.344,-178.599,6.668,148.814
C01065=1161.956,144.809,-56.365,-178.597,6.670,148.814
C01066=1161.951,145.058,-56.385,-178.594,6.671,148.814
C01067=1161.946,145.307,-56.406,-178.591,6.673,148.813
C01068=1161.942,145.556,-56.427,-178.589,6.675,148.813
C01069=1161.937,145.806,-56.448,-178.586,6.677,148.812
C01070=1161.933,146.055,-56.468,-178.583,6.678,148.812
C01071=1161.928,146.303,-56.490,-178.581,6.680,148.812
C01072=1161.923,146.552,-56.510,-178.578,6.682,148.811
C01073=1161.918,146.802,-56.531,-178.575,6.684,148.811
C01074=1161.914,147.050,-56.552,-178.572,6.685,148.810
C01075=1161.909,147.300,-56.573,-178.570,6.687,148.810
C01076=1161.904,147.548,-56.594,-178.567,6.689,148.810
C01077=1161.899,147.797,-56.615,-178.564,6.691,148.809
C01078=1161.894,148.047,-56.636,-178.562,6.692,148.809
C01079=1161.890,148.296,-56.656,-178.559,6.694,148.809
C01080=1161.885,148.546,-56.677,-178.556,6.696,148.808
C01081=1161.880,148.794,-56.699,-178.554,6.697,148.808
C01082=1161.876,149.043,-56.719,-178.551,6.699,148.807
C01083=1161.871,149.292,-56.740,-178.548,6.701,148.807
C01084=1161.866,149.541,-56.761,-178.545,6.703,148.807
C01085=1161.861,149.790,-56.782,-178.543,6.704,148.806
C01086=1161.857,150.040,-56.804,-178.539,6.707,148.806
C01087=1161.853,150.288,-56.825,-178.537,6.709,148.806
C01088=1161.847,150.537,-56.846,-178.534,6.710,148.805
C01089=1161.842,150.787,-56.867,-178.531,6.712,148.805
C01090=1161.838,151.035,-56.888,-178.529,6.714,148.804
C01091=1161.833,151.284,-56.909,-178.526,6.716,148.804
C01092=1161.828,151.534,-56.930,-178.523,6.717,148.804
C01093=1161.824,151.783,-56.951,-178.521,6.719,148.803
C01094=1161.819,152.032,-56.972,-178.518,6.721,148.803
C01095=1161.814,152.281,-56.994,-178.516,6.723,148.803
C01096=1161.809,152.530,-57.015,-178.513,6.725,148.802
C01097=1161.805,152.779,-57.036,-178.510,6.726,148.802
C01098=1161.800,153.028,-57.057,-178.508,6.728,148.802
C01099=1161.795,153.277,-57.078,-178.504,6.731,148.801
C01100=1161.790,153.526,-57.100,-178.502,6.732,148.801
C01101=1161.786,153.776,-57.121,-178.499,6.734,148.800
C01102=1161.782,154.024,-57.142,-178.496,6.736,148.800
C01103=1161.776,154.274,-57.163,-178.493,6.738,148.800
C01104=1161.771,154.522,-57.185,-178.491,6.739,148.799
C01105=1161.767,154.772,-57.206,-178.488,6.741,148.799
C01106=1161.763,155.020,-57.227,-178.485,6.743,148.799
C01107=1161.758,155.270,-57.248,-178.483,6.745,148.798
C01108=1161.753,155.518,-57.270,-178.480,6.746,148.798
C01109=1161.748,155.768,-57.292,-178.477,6.749,148.797
C01110=1161.743,156.017,-57.313,-178.474,6.751,148.797
C01111=1161.739,156.265,-57.334,-178.471,6.752,148.797
C01112=1161.734,156.515,-57.355,-178.469,6.754,148.796
C01113=1161.730,156.764,-57.377,-178.466,6.756,148.796
C01114=1161.725,157.013,-57.399,-178.464,6.758,148.796
C01115=1161.720,157.262,-57.420,-178.461,6.760,148.795
C01116=1161.715,157.511,-57.442,-178.458,6.761,148.795
C01117=1161.711,157.780,-57.465,-178.455,6.764,148.795
C01118=1161.705,158.049,-57.488,-178.452,6.766,148.794
C01119=1161.700,158.317,-57.511,-178.449,6.767,148.794
C01120=1161.695,158.587,-57.535,-178.446,6.770,148.793
C01121=1161.690,158.836,-57.557,-178.443,6.771,148.793
C01122=1161.685,159.085,-57.578,-178.441,6.774,148.793
C01123=1161.680,159.334,-57.599,-178.438,6.775,148.792
C01124=1161.677,159.583,-57.621,-178.436,6.777,148.792
C01125=1161.672,159.832,-57.642,-178.432,6.780,148.792
C01126=1161.667,160.081,-57.663,-178.430,6.781,148.791
C01127=1161.662,160.330,-57.685,-178.427,6.783,148.791
C01128=1161.658,160.579,-57.707,-178.424,6.785,148.791
C01129=1161.653,160.828,-57.729,-178.421,6.787,148.790
C01130=1161.648,161.077,-57.751,-178.419,6.788,148.790
C01131=1161.644,161.325,-57.772,-178.416,6.790,148.789
C01132=1161.639,161.575,-57.794,-178.413,6.793,148.789
C01133=1161.634,161.824,-57.815,-178.411,6.795,148.789
C01134=1161.629,162.073,-57.837,-178.408,6.796,148.789
C01135=1161.625,162.322,-57.859,-178.405,6.798,148.788
C01136=1161.620,162.571,-57.881,-178.403,6.800,148.788
C01137=1161.616,162.820,-57.903,-178.400,6.802,148.787
C01138=1161.611,163.069,-57.925,-178.397,6.803,148.787
C01139=1161.607,163.318,-57.947,-178.394,6.806,148.787
C01140=1161.601,163.567,-57.969,-178.391,6.808,148.786
C01141=1161.596,163.816,-57.990,-178.388,6.809,148.786
C01142=1161.592,164.065,-58.012,-178.386,6.812,148.786
C01143=1161.587,164.314,-58.034,-178.384,6.813,148.785
C01144=1161.583,164.563,-58.056,-178.381,6.815,148.785
C01145=1161.578,164.812,-58.077,-178.378,6.818,148.785
C01146=1161.573,165.061,-58.099,-178.375,6.819,148.784
C01147=1161.569,165.310,-58.121,-178.372,6.821,148.784
C01148=1161.564,165.559,-58.143,-178.370,6.823,148.784
C01149=1161.559,165.808,-58.165,-178.367,6.825,148.783
C01150=1161.554,166.058,-58.187,-178.364,6.828,148.783
C01151=1161.550,166.306,-58.210,-178.361,6.829,148.783
C01152=1161.546,166.555,-58.232,-178.359,6.831,148.782
C01153=1161.541,166.804,-58.254,-178.356,6.833,148.782
C01154=1161.536,167.053,-58.276,-178.353,6.834,148.782
C01155=1161.532,167.302,-58.297,-178.351,6.836,148.781
C01156=1161.527,167.551,-58.320,-178.348,6.839,148.781
C01157=1161.522,167.800,-58.342,-178.345,6.841,148.781
C01158=1161.517,168.049,-58.364,-178.342,6.843,148.780
C01159=1161.513,168.298,-58.385,-178.340,6.844,148.780
C01160=1161.509,168.547,-58.408,-178.337,6.846,148.780
C01161=1161.503,168.796,-58.430,-178.334,6.849,148.779
C01162=1161.499,169.045,-58.452,-178.331,6.850,148.779
C01163=1161.494,169.294,-58.474,-178.329,6.853,148.779
C01164=1161.490,169.543,-58.496,-178.326,6.854,148.778
C01165=1161.484,169.791,-58.519,-178.323,6.857,148.778
C01166=1161.480,170.041,-58.541,-178.320,6.859,148.778
C01167=1161.475,170.289,-58.563,-178.317,6.860,148.777
C01168=1161.471,170.539,-58.585,-178.315,6.862,148.777
C01169=1161.466,170.788,-58.608,-178.313,6.864,148.777
C01170=1161.461,171.036,-58.630,-178.309,6.867,148.776
C01171=1161.457,171.286,-58.652,-178.307,6.869,148.776
C01172=1161.451,171.535,-58.674,-178.304,6.870,148.776
C01173=1161.447,171.783,-58.697,-178.301,6.872,148.775
C01174=1161.443,172.032,-58.719,-178.298,6.875,148.775
C01175=1161.438,172.282,-58.741,-178.296,6.877,148.775
C01176=1161.434,172.530,-58.764,-178.293,6.878,148.775
C01177=1161.429,172.779,-58.786,-178.290,6.880,148.774
C01178=1161.424,173.029,-58.809,-178.288,6.882,148.774
C01179=1161.420,173.277,-58.831,-178.284,6.885,148.773
C01180=1161.414,173.526,-58.854,-178.282,6.887,148.773
C01181=1161.410,173.775,-58.876,-178.280,6.888,148.773
C01182=1161.405,174.024,-58.898,-178.277,6.890,148.773
C01183=1161.401,174.273,-58.921,-178.274,6.893,148.772
C01184=1161.396,174.522,-58.943,-178.271,6.894,148.772
C01185=1161.391,174.771,-58.966,-178.269,6.897,148.772
C01186=1161.387,175.020,-58.988,-178.266,6.898,148.771
C01187=1161.383,175.269,-59.011,-178.263,6.901,148.771
C01188=1161.377,175.517,-59.034,-178.260,6.903,148.771
C01189=1161.373,175.767,-59.056,-178.258,6.905,148.770
C01190=1161.368,176.016,-59.079,-178.255,6.906,148.770
C01191=1161.363,176.264,-59.101,-178.252,6.909,148.770
C01192=1161.359,176.513,-59.124,-178.249,6.911,148.769
C01193=1161.354,176.763,-59.146,-178.246,6.913,148.769
C01194=1161.349,177.011,-59.169,-178.244,6.915,148.769
C01195=1161.345,177.260,-59.192,-178.241,6.917,148.769
C01196=1161.340,177.509,-59.214,-178.238,6.919,148.768
C01197=1161.336,177.758,-59.237,-178.236,6.921,148.768
C01198=1161.331,178.007,-59.259,-178.233,6.924,148.768
C01199=1161.327,178.256,-59.282,-178.230,6.925,148.767
C01200=1161.322,178.505,-59.306,-178.227,6.927,148.767
C01201=1161.317,178.754,-59.327,-178.225,6.929,148.767
C01202=1161.312,179.003,-59.351,-178.221,6.931,148.766
C01203=1161.308,179.251,-59.373,-178.219,6.934,148.766
C01204=1161.303,179.501,-59.396,-178.217,6.935,148.766
C01205=1161.299,179.749,-59.418,-178.214,6.937,148.765
C01206=1161.294,179.998,-59.442,-178.211,6.940,148.765
C01207=1161.289,180.248,-59.464,-178.208,6.942,148.765
C01208=1161.285,180.496,-59.487,-178.206,6.944,148.765
C01209=1161.281,180.745,-59.511,-178.202,6.946,148.764
C01210=1161.276,180.993,-59.533,-178.200,6.948,148.764
C01211=1161.271,181.243,-59.556,-178.198,6.950,148.764
C01212=1161.266,181.492,-59.579,-178.195,6.952,148.763
C01213=1161.262,181.741,-59.602,-178.192,6.954,148.763
C01214=1161.257,181.989,-59.625,-178.189,6.956,148.763
C01215=1161.252,182.238,-59.648,-178.187,6.958,148.763
C01216=1161.248,182.488,-59.670,-178.183,6.961,148.762
C01217=1161.243,182.737,-59.693,-178.181,6.962,148.762
C01218=1161.239,182.985,-59.716,-178.179,6.965,148.762
C01219=1161.235,183.234,-59.740,-178.175,6.967,148.761
C01220=1161.229,183.483,-59.763,-178.173,6.969,148.761
C01221=1161.224,183.752,-59.788,-178.169,6.971,148.761
C01222=1161.219,184.022,-59.812,-178.167,6.973,148.760
C01223=1161.215,184.292,-59.837,-178.163,6.976,148.760
C01224=1161.209,184.562,-59.862,-178.161,6.978,148.760
C01225=1161.205,184.810,-59.885,-178.158,6.980,148.759
C01226=1161.200,185.059,-59.908,-178.155,6.982,148.759
C01227=1161.195,185.308,-59.932,-178.153,6.984,148.759
C01228=1161.191,185.557,-59.955,-178.150,6.987,148.759
C01229=1161.187,185.806,-59.978,-178.147,6.989,148.758
C01230=1161.182,186.055,-60.001,-178.144,6.990,148.758
C01231=1161.177,186.304,-60.024,-178.142,6.993,148.758
C01232=1161.173,186.553,-60.048,-178.139,6.995,148.757
C01233=1161.168,186.801,-60.070,-178.136,6.997,148.757
C01234=1161.163,187.050,-60.094,-178.133,7.000,148.757
C01235=1161.159,187.299,-60.117,-178.131,7.002,148.757
C01236=1161.154,187.548,-60.140,-178.128,7.003,148.756
C01237=1161.149,187.797,-60.164,-178.125,7.006,148.756
C01238=1161.145,188.046,-60.188,-178.123,7.008,148.756
C01239=1161.141,188.294,-60.210,-178.120,7.010,148.755
C01240=1161.136,188.543,-60.234,-178.117,7.012,148.755
C01241=1161.132,188.792,-60.257,-178.114,7.014,148.755
C01242=1161.127,189.041,-60.281,-178.112,7.016,148.755
C01243=1161.122,189.290,-60.304,-178.109,7.019,148.754
C01244=1161.117,189.539,-60.327,-178.106,7.021,148.754
C01245=1161.113,189.789,-60.351,-178.104,7.023,148.754
C01246=1161.108,190.036,-60.374,-178.100,7.025,148.753
C01247=1161.103,190.285,-60.398,-178.098,7.027,148.753
C01248=1161.099,190.534,-60.420,-178.095,7.030,148.753
C01249=1161.094,190.783,-60.444,-178.092,7.032,148.753
C01250=1161.090,191.032,-60.467,-178.090,7.034,148.753
C01251=1161.085,191.280,-60.491,-178.087,7.036,148.752
C01252=1161.081,191.529,-60.515,-178.084,7.038,148.752
C01253=1161.076,191.779,-60.538,-178.082,7.040,148.752
C01254=1161.071,192.028,-60.561,-178.079,7.043,148.751
C01255=1161.067,192.276,-60.585,-178.076,7.045,148.751
C01256=1161.062,192.525,-60.609,-178.073,7.047,148.751
C01257=1161.057,192.774,-60.632,-178.070,7.049,148.751
C01258=1161.053,193.022,-60.656,-178.068,7.051,148.750
C01259=1161.048,193.271,-60.680,-178.065,7.054,148.750
C01260=1161.044,193.521,-60.703,-178.062,7.056,148.750
C01261=1161.039,193.769,-60.727,-178.060,7.058,148.750
C01262=1161.035,194.018,-60.750,-178.057,7.060,148.749
C01263=1161.030,194.267,-60.774,-178.054,7.062,148.749
C01264=1161.025,194.515,-60.798,-178.051,7.065,148.749
C01265=1161.021,194.765,-60.822,-178.049,7.067,148.748
C01266=1161.017,195.014,-60.846,-178.046,7.069,148.748
C01267=1161.012,195.263,-60.869,-178.043,7.072,148.748
C01268=1161.007,195.511,-60.894,-178.041,7.073,148.748
C01269=1161.002,195.760,-60.917,-178.038,7.076,148.748
C01270=1160.998,196.009,-60.941,-178.035,7.078,148.747
C01271=1160.993,196.258,-60.964,-178.032,7.080,148.747
C01272=1160.989,196.507,-60.988,-178.030,7.083,148.747
C01273=1160.984,196.755,-61.012,-178.027,7.084,148.746
C01274=1160.980,197.004,-61.036,-178.024,7.087,148.746
C01275=1160.975,197.253,-61.059,-178.021,7.089,148.746
C01276=1160.971,197.501,-61.083,-178.019,7.091,148.746
C01277=1160.966,197.751,-61.108,-178.016,7.094,148.745
C01278=1160.962,198.000,-61.132,-178.013,7.096,148.745
C01279=1160.957,198.249,-61.155,-178.010,7.098,148.745
C01280=1160.952,198.497,-61.179,-178.008,7.100,148.745
C01281=1160.948,198.746,-61.203,-178.005,7.103,148.744
C01282=1160.943,198.994,-61.227,-178.002,7.105,148.744
C01283=1160.938,199.243,-61.251,-178.000,7.107,148.744
C01284=1160.934,199.493,-61.275,-177.997,7.110,148.744
C01285=1160.930,199.741,-61.299,-177.994,7.111,148.743
C01286=1160.925,199.990,-61.323,-177.991,7.114,148.743
C01287=1160.921,200.239,-61.347,-177.989,7.116,148.743
C01288=1160.915,200.487,-61.371,-177.986,7.119,148.743
C01289=1160.911,200.736,-61.395,-177.983,7.121,148.742
C01290=1160.907,200.986,-61.419,-177.981,7.123,148.742
C01291=1160.903,201.234,-61.443,-177.977,7.125,148.742
C01292=1160.897,201.483,-61.468,-177.975,7.127,148.742
C01293=1160.893,201.731,-61.492,-177.972,7.130,148.741
C01294=1160.888,201.980,-61.515,-177.970,7.132,148.741
C01295=1160.884,202.230,-61.540,-177.966,7.135,148.741
C01296=1160.879,202.478,-61.564,-177.964,7.137,148.741
C01297=1160.875,202.726,-61.588,-177.961,7.139,148.740
C01298=1160.871,202.975,-61.612,-177.958,7.141,148.740
C01299=1160.865,203.224,-61.636,-177.956,7.144,148.740
C01300=1160.861,203.473,-61.661,-177.953,7.146,148.740
C01301=1160.857,203.722,-61.685,-177.951,7.148,148.740
C01302=1160.852,203.970,-61.710,-177.947,7.150,148.739
C01303=1160.847,204.219,-61.734,-177.945,7.153,148.739
C01304=1160.843,204.468,-61.759,-177.942,7.155,148.739
C01305=1160.839,204.717,-61.783,-177.940,7.157,148.739
C01306=1160.834,204.965,-61.807,-177.937,7.160,148.738
C01307=1160.829,205.214,-61.831,-177.934,7.162,148.738
C01308=1160.825,205.464,-61.855,-177.931,7.164,148.738
C01309=1160.820,205.712,-61.880,-177.928,7.166,148.738
C01310=1160.815,205.961,-61.904,-177.926,7.169,148.737
C01311=1160.812,206.210,-61.928,-177.923,7.171,148.737
C01312=1160.806,206.459,-61.953,-177.920,7.174,148.737
C01313=1160.802,206.707,-61.977,-177.917,7.176,148.737
C01314=1160.797,206.956,-62.002,-177.915,7.179,148.737
C01315=1160.793,207.205,-62.026,-177.912,7.180,148.736
C01316=1160.788,207.454,-62.051,-177.909,7.183,148.736
C01317=1160.784,207.702,-62.075,-177.907,7.185,148.736
C01318=1160.779,207.951,-62.100,-177.904,7.188,148.736
C01319=1160.775,208.200,-62.124,-177.901,7.190,148.735
C01320=1160.770,208.448,-62.149,-177.898,7.193,148.735
C01321=1160.766,208.697,-62.174,-177.896,7.194,148.735
C01322=1160.761,208.946,-62.199,-177.893,7.197,148.735
C01323=1160.757,209.194,-62.223,-177.890,7.199,148.734
C01324=1160.752,209.444,-62.248,-177.887,7.202,148.734
C01325=1160.747,209.714,-62.274,-177.885,7.204,148.734
C01326=1160.742,209.984,-62.301,-177.881,7.206,148.734
C01327=1160.737,210.255,-62.328,-177.879,7.209,148.734
C01328=1160.732,210.525,-62.355,-177.875,7.212,148.733
C01329=1160.728,210.774,-62.379,-177.873,7.214,148.733
C01330=1160.723,211.023,-62.404,-177.870,7.217,148.733
C01331=1160.718,211.271,-62.429,-177.868,7.219,148.733
C01332=1160.714,211.520,-62.454,-177.865,7.221,148.732
C01333=1160.709,211.769,-62.479,-177.862,7.224,148.732
C01334=1160.706,212.018,-62.503,-177.859,7.226,148.732
C01335=1160.700,212.267,-62.528,-177.857,7.228,148.732
C01336=1160.696,212.515,-62.553,-177.854,7.231,148.732
C01337=1160.692,212.764,-62.577,-177.851,7.234,148.731
C01338=1160.687,213.012,-62.602,-177.848,7.236,148.731
C01339=1160.682,213.262,-62.627,-177.845,7.238,148.731
C01340=1160.678,213.510,-62.652,-177.843,7.241,148.731
C01341=1160.674,213.759,-62.677,-177.840,7.243,148.731
C01342=1160.669,214.007,-62.702,-177.838,7.245,148.730
C01343=1160.665,214.256,-62.727,-177.835,7.248,148.730
C01344=1160.660,214.505,-62.751,-177.832,7.250,148.730
C01345=1160.656,214.754,-62.777,-177.829,7.253,148.730
C01346=1160.651,215.002,-62.801,-177.827,7.255,148.730
C01347=1160.646,215.251,-62.826,-177.824,7.257,148.729
C01348=1160.642,215.500,-62.852,-177.821,7.259,148.729
C01349=1160.637,215.749,-62.876,-177.818,7.262,148.729
C01350=1160.633,215.997,-62.902,-177.815,7.265,148.729
C01351=1160.628,216.246,-62.926,-177.813,7.267,148.729
C01352=1160.624,216.495,-62.952,-177.810,7.270,148.728
C01353=1160.619,216.743,-62.977,-177.808,7.272,148.728
C01354=1160.615,216.992,-63.002,-177.804,7.274,148.728
C01355=1160.610,217.240,-63.026,-177.802,7.276,148.728
C01356=1160.606,217.489,-63.052,-177.799,7.279,148.727
C01357=1160.601,217.738,-63.077,-177.796,7.282,148.727
C01358=1160.597,217.987,-63.103,-177.794,7.284,148.727
C01359=1160.593,218.235,-63.128,-177.791,7.287,148.727
C01360=1160.588,218.484,-63.152,-177.789,7.289,148.727
C01361=1160.584,218.733,-63.178,-177.785,7.291,148.727
C01362=1160.579,218.982,-63.203,-177.783,7.294,148.726
C01363=1160.574,219.230,-63.229,-177.780,7.296,148.726
C01364=1160.569,219.478,-63.254,-177.777,7.299,148.726
C01365=1160.566,219.728,-63.278,-177.775,7.301,148.726
C01366=1160.561,219.976,-63.304,-177.772,7.304,148.726
C01367=1160.557,220.224,-63.330,-177.770,7.306,148.725
C01368=1160.552,220.474,-63.355,-177.766,7.308,148.725
C01369=1160.547,220.722,-63.380,-177.764,7.311,148.725
C01370=1160.543,220.971,-63.406,-177.761,7.314,148.725
C01371=1160.538,221.220,-63.430,-177.758,7.316,148.725
C01372=1160.534,221.468,-63.456,-177.756,7.318,148.725
C01373=1160.529,221.717,-63.482,-177.753,7.321,148.724
C01374=1160.525,221.965,-63.507,-177.750,7.323,148.724
C01375=1160.520,222.215,-63.532,-177.748,7.326,148.724
C01376=1160.515,222.463,-63.558,-177.744,7.328,148.724
C01377=1160.511,222.712,-63.583,-177.742,7.331,148.724
C01378=1160.507,222.960,-63.609,-177.739,7.333,148.723
C01379=1160.502,223.209,-63.635,-177.736,7.336,148.723
C01380=1160.497,223.458,-63.660,-177.734,7.338,148.723
C01381=1160.493,223.707,-63.685,-177.731,7.341,148.723
C01382=1160.488,223.955,-63.711,-177.729,7.343,148.723
C01383=1160.484,224.204,-63.737,-177.726,7.346,148.723
C01384=1160.480,224.452,-63.762,-177.722,7.349,148.722
C01385=1160.475,224.701,-63.788,-177.720,7.351,148.722
C01386=1160.471,224.949,-63.813,-177.718,7.354,148.722
C01387=1160.467,225.198,-63.839,-177.715,7.355,148.722
C01388=1160.462,225.447,-63.864,-177.712,7.358,148.722
C01389=1160.457,225.696,-63.890,-177.709,7.361,148.721
C01390=1160.453,225.945,-63.915,-177.707,7.363,148.721
C01391=1160.448,226.193,-63.941,-177.704,7.366,148.721
C01392=1160.444,226.441,-63.966,-177.701,7.369,148.721
C01393=1160.440,226.690,-63.992,-177.698,7.371,148.721
C01394=1160.436,226.939,-64.018,-177.696,7.374,148.721
C01395=1160.431,227.187,-64.043,-177.692,7.376,148.720
C01396=1160.426,227.436,-64.070,-177.690,7.378,148.720
C01397=1160.422,227.685,-64.095,-177.687,7.381,148.720
C01398=1160.417,227.933,-64.121,-177.684,7.384,148.720
C01399=1160.413,228.181,-64.147,-177.682,7.386,148.720
C01400=1160.409,228.430,-64.173,-177.679,7.389,148.720
C01401=1160.404,228.679,-64.199,-177.677,7.391,148.719
C01402=1160.399,228.927,-64.225,-177.674,7.394,148.719
C01403=1160.395,229.176,-64.251,-177.671,7.397,148.719
C01404=1160.390,229.425,-64.276,-177.668,7.398,148.719
C01405=1160.386,229.674,-64.302,-177.666,7.401,148.719
C01406=1160.382,229.923,-64.328,-177.663,7.404,148.719
C01407=1160.377,230.170,-64.355,-177.660,7.406,148.718
C01408=1160.372,230.419,-64.380,-177.657,7.409,148.718
C01409=1160.368,230.668,-64.406,-177.655,7.412,148.718
C01410=1160.364,230.917,-64.432,-177.652,7.414,148.718
C01411=1160.359,231.166,-64.458,-177.649,7.417,148.718
C01412=1160.355,231.413,-64.484,-177.646,7.420,148.718
C01413=1160.350,231.662,-64.510,-177.644,7.422,148.718
C01414=1160.346,231.911,-64.536,-177.641,7.424,148.717
C01415=1160.341,232.160,-64.562,-177.638,7.427,148.717
C01416=1160.337,232.408,-64.589,-177.635,7.430,148.717
C01417=1160.332,232.656,-64.614,-177.633,7.432,148.717
C01418=1160.327,232.906,-64.640,-177.630,7.435,148.717
C01419=1160.324,233.154,-64.667,-177.627,7.438,148.717
C01420=1160.319,233.402,-64.692,-177.625,7.440,148.717
C01421=1160.314,233.652,-64.719,-177.622,7.443,148.716
C01422=1160.310,233.900,-64.745,-177.619,7.445,148.716
C01423=1160.306,234.149,-64.771,-177.617,7.448,148.716
C01424=1160.301,234.396,-64.798,-177.614,7.451,148.716
C01425=1160.297,234.645,-64.823,-177.611,7.453,148.716
C01426=1160.292,234.894,-64.849,-177.609,7.455,148.716
C01427=1160.288,235.142,-64.876,-177.606,7.458,148.715
C01428=1160.284,235.391,-64.902,-177.603,7.461,148.715
C01429=1160.278,235.663,-64.931,-177.600,7.464,148.715
C01430=1160.274,235.935,-64.959,-177.597,7.467,148.715
C01431=1160.269,236.206,-64.989,-177.594,7.469,148.715
C01432=1160.264,236.478,-65.018,-177.591,7.472,148.715
C01433=1160.259,236.727,-65.044,-177.588,7.475,148.715
C01434=1160.255,236.975,-65.070,-177.585,7.478,148.714
C01435=1160.251,237.224,-65.096,-177.583,7.480,148.714
C01436=1160.246,237.472,-65.123,-177.580,7.483,148.714
C01437=1160.242,237.721,-65.149,-177.577,7.486,148.714
C01438=1160.238,237.970,-65.176,-177.575,7.488,148.714
C01439=1160.233,238.218,-65.202,-177.572,7.491,148.714
C01440=1160.229,238.467,-65.229,-177.569,7.493,148.714
C01441=1160.225,238.715,-65.255,-177.566,7.496,148.713
C01442=1160.220,238.964,-65.282,-177.564,7.499,148.713
C01443=1160.215,239.212,-65.308,-177.561,7.501,148.713
C01444=1160.211,239.460,-65.335,-177.558,7.504,148.713
C01445=1160.206,239.709,-65.361,-177.555,7.507,148.713
C01446=1160.202,239.957,-65.388,-177.553,7.509,148.713
C01447=1160.197,240.206,-65.415,-177.550,7.512,148.713
C01448=1160.193,240.455,-65.440,-177.547,7.515,148.712
C01449=1160.188,240.703,-65.467,-177.544,7.518,148.712
C01450=1160.184,240.951,-65.494,-177.542,7.520,148.712
C01451=1160.180,241.200,-65.521,-177.539,7.523,148.712
C01452=1160.175,241.449,-65.547,-177.537,7.526,148.712
C01453=1160.171,241.697,-65.574,-177.533,7.528,148.712
C01454=1160.167,241.946,-65.601,-177.531,7.530,148.712
C01455=1160.163,242.195,-65.628,-177.528,7.533,148.712
C01456=1160.158,242.444,-65.654,-177.526,7.536,148.712
C01457=1160.153,242.692,-65.681,-177.523,7.539,148.712
C01458=1160.149,242.940,-65.708,-177.520,7.541,148.711
C01459=1160.145,243.189,-65.735,-177.517,7.544,148.711
C01460=1160.140,243.437,-65.762,-177.515,7.547,148.711
C01461=1160.136,243.686,-65.788,-177.512,7.550,148.711
C01462=1160.131,243.934,-65.815,-177.510,7.552,148.711
C01463=1160.126,244.183,-65.842,-177.507,7.555,148.711
C01464=1160.123,244.431,-65.868,-177.504,7.558,148.711
C01465=1160.118,244.680,-65.895,-177.501,7.560,148.710
C01466=1160.113,244.928,-65.922,-177.499,7.563,148.710
C01467=1160.109,245.177,-65.949,-177.496,7.566,148.710
C01468=1160.105,245.426,-65.976,-177.493,7.568,148.710
C01469=1160.101,245.674,-66.003,-177.490,7.571,148.710
C01470=1160.096,245.923,-66.030,-177.488,7.574,148.710
C01471=1160.091,246.171,-66.057,-177.485,7.576,148.710
C01472=1160.087,246.419,-66.084,-177.482,7.579,148.710
C01473=1160.083,246.668,-66.111,-177.479,7.582,148.710
C01474=1160.078,246.916,-66.138,-177.477,7.585,148.710
C01475=1160.073,247.165,-66.165,-177.474,7.587,148.709
C01476=1160.069,247.414,-66.192,-177.472,7.590,148.709
C01477=1160.065,247.662,-66.219,-177.469,7.593,148.709
C01478=1160.061,247.910,-66.247,-177.466,7.596,148.709
C01479=1160.056,248.159,-66.274,-177.463,7.599,148.709
C01480=1160.052,248.407,-66.301,-177.461,7.601,148.709
C01481=1160.047,248.656,-66.328,-177.458,7.604,148.709
C01482=1160.042,248.904,-66.355,-177.455,7.607,148.709
C01483=1160.038,249.153,-66.382,-177.452,7.610,148.709
C01484=1160.034,249.402,-66.409,-177.450,7.612,148.709
C01485=1160.030,249.649,-66.436,-177.448,7.615,148.708
C01486=1160.025,249.898,-66.464,-177.444,7.617,148.708
C01487=1160.021,250.146,-66.491,-177.442,7.620,148.708
C01488=1160.017,250.396,-66.518,-177.439,7.623,148.708
C01489=1160.012,250.644,-66.545,-177.436,7.626,148.708
C01490=1160.008,250.892,-66.573,-177.433,7.629,148.708
C01491=1160.003,251.140,-66.600,-177.431,7.631,148.708
C01492=1159.999,251.390,-66.627,-177.428,7.634,148.708
C01493=1159.995,251.638,-66.655,-177.425,7.637,148.708
C01494=1159.990,251.886,-66.682,-177.423,7.640,148.708
C01495=1159.985,252.135,-66.709,-177.420,7.643,148.708
C01496=1159.981,252.384,-66.737,-177.418,7.645,148.707
C01497=1159.977,252.632,-66.764,-177.415,7.648,148.707
C01498=1159.972,252.880,-66.791,-177.412,7.651,148.707
C01499=1159.968,253.128,-66.819,-177.409,7.654,148.707
C01500=1159.964,253.377,-66.847,-177.406,7.656,148.707
C01501=1159.959,253.626,-66.874,-177.403,7.659,148.707
C01502=1159.955,253.874,-66.902,-177.401,7.662,148.707
C01503=1159.950,254.122,-66.929,-177.398,7.665,148.707
C01504=1159.946,254.371,-66.957,-177.396,7.667,148.707
C01505=1159.942,254.619,-66.984,-177.393,7.670,148.707
C01506=1159.937,254.867,-67.012,-177.390,7.673,148.707
C01507=1159.933,255.116,-67.039,-177.387,7.676,148.707
C01508=1159.929,255.365,-67.066,-177.385,7.678,148.706
C01509=1159.924,255.613,-67.094,-177.382,7.681,148.706
C01510=1159.920,255.862,-67.121,-177.380,7.684,148.706
C01511=1159.916,256.110,-67.149,-177.377,7.687,148.706
C01512=1159.912,256.357,-67.177,-177.374,7.690,148.706
C01513=1159.907,256.607,-67.205,-177.371,7.693,148.706
C01514=1159.902,256.855,-67.233,-177.369,7.696,148.706
C01515=1159.898,257.103,-67.260,-177.366,7.698,148.706
C01516=1159.894,257.352,-67.288,-177.364,7.701,148.706
C01517=1159.889,257.600,-67.315,-177.361,7.704,148.706
C01518=1159.885,257.848,-67.343,-177.358,7.707,148.706
C01519=1159.881,258.097,-67.371,-177.355,7.710,148.706
C01520=1159.876,258.346,-67.398,-177.352,7.713,148.705
C01521=1159.872,258.594,-67.426,-177.349,7.716,148.705
C01522=1159.868,258.842,-67.454,-177.347,7.718,148.705
C01523=1159.863,259.091,-67.481,-177.344,7.721,148.705
C01524=1159.859,259.339,-67.510,-177.342,7.724,148.705
C01525=1159.854,259.587,-67.538,-177.339,7.727,148.705
C01526=1159.850,259.835,-67.566,-177.336,7.730,148.705
C01527=1159.846,260.084,-67.593,-177.333,7.732,148.705
C01528=1159.842,260.332,-67.621,-177.331,7.735,148.705
C01529=1159.837,260.581,-67.650,-177.328,7.739,148.705
C01530=1159.833,260.829,-67.677,-177.326,7.741,148.705
C01531=1159.829,261.078,-67.705,-177.323,7.744,148.705
C01532=1159.824,261.326,-67.733,-177.321,7.747,148.705
C01533=1159.819,261.600,-67.764,-177.317,7.749,148.705
C01534=1159.814,261.873,-67.795,-177.314,7.753,148.705
C01535=1159.810,262.146,-67.826,-177.311,7.756,148.705
C01536=1159.805,262.419,-67.857,-177.308,7.759,148.704
C01537=1159.801,262.667,-67.884,-177.306,7.762,148.704
C01538=1159.796,262.917,-67.912,-177.303,7.765,148.704
C01539=1159.792,263.164,-67.940,-177.300,7.768,148.704
C01540=1159.788,263.413,-67.968,-177.297,7.771,148.704
C01541=1159.783,263.661,-67.997,-177.295,7.774,148.704
C01542=1159.779,263.910,-68.025,-177.292,7.777,148.704
C01543=1159.774,264.158,-68.053,-177.290,7.780,148.704
C01544=1159.770,264.407,-68.081,-177.287,7.782,148.704
C01545=1159.766,264.654,-68.109,-177.285,7.785,148.704
C01546=1159.761,264.903,-68.138,-177.282,7.788,148.704
C01547=1159.757,265.151,-68.166,-177.279,7.791,148.704
C01548=1159.753,265.400,-68.194,-177.276,7.794,148.704
C01549=1159.748,265.648,-68.222,-177.274,7.797,148.704
C01550=1159.744,265.897,-68.251,-177.271,7.800,148.704
C01551=1159.739,266.145,-68.279,-177.268,7.803,148.704
C01552=1159.735,266.394,-68.307,-177.265,7.806,148.704
C01553=1159.731,266.642,-68.335,-177.263,7.809,148.704
C01554=1159.727,266.890,-68.363,-177.260,7.812,148.704
C01555=1159.722,267.138,-68.393,-177.258,7.814,148.704
C01556=1159.718,267.386,-68.421,-177.255,7.817,148.704
C01557=1159.714,267.635,-68.449,-177.253,7.820,148.704
C01558=1159.709,267.883,-68.477,-177.250,7.823,148.704
C01559=1159.705,268.132,-68.506,-177.247,7.826,148.704
C01560=1159.700,268.380,-68.534,-177.244,7.829,148.703
C01561=1159.696,268.628,-68.563,-177.241,7.832,148.703
C01562=1159.691,268.876,-68.592,-177.239,7.835,148.703
C01563=1159.688,269.125,-68.620,-177.236,7.838,148.703
C01564=1159.683,269.374,-68.648,-177.233,7.841,148.703
C01565=1159.679,269.622,-68.676,-177.230,7.844,148.703
C01566=1159.675,269.870,-68.706,-177.228,7.847,148.703
C01567=1159.670,270.119,-68.734,-177.225,7.850,148.703
C01568=1159.666,270.367,-68.762,-177.223,7.852,148.703
C01569=1159.662,270.615,-68.792,-177.220,7.855,148.703
C01570=1159.657,270.863,-68.819,-177.218,7.858,148.703
C01571=1159.653,271.112,-68.848,-177.215,7.861,148.703
C01572=1159.649,271.360,-68.878,-177.212,7.864,148.703
C01573=1159.644,271.608,-68.905,-177.209,7.867,148.703
C01574=1159.640,271.857,-68.934,-177.207,7.870,148.703
C01575=1159.636,272.105,-68.964,-177.204,7.873,148.703
C01576=1159.631,272.353,-68.991,-177.202,7.876,148.703
C01577=1159.627,272.602,-69.020,-177.199,7.879,148.703
C01578=1159.623,272.850,-69.049,-177.196,7.882,148.703
C01579=1159.618,273.098,-69.077,-177.193,7.885,148.703
C01580=1159.614,273.346,-69.107,-177.190,7.888,148.703
C01581=1159.610,273.595,-69.135,-177.188,7.891,148.703
C01582=1159.606,273.843,-69.164,-177.185,7.894,148.703
C01583=1159.601,274.091,-69.193,-177.183,7.897,148.703
C01584=1159.597,274.339,-69.222,-177.180,7.900,148.703
C01585=1159.592,274.588,-69.251,-177.177,7.903,148.703
C01586=1159.588,274.836,-69.279,-177.174,7.906,148.703
C01587=1159.584,275.084,-69.308,-177.172,7.909,148.703
C01588=1159.580,275.333,-69.338,-177.169,7.912,148.703
C01589=1159.575,275.582,-69.366,-177.167,7.915,148.703
C01590=1159.571,275.829,-69.395,-177.164,7.917,148.703
C01591=1159.567,276.077,-69.424,-177.162,7.920,148.703
C01592=1159.562,276.326,-69.453,-177.159,7.923,148.703
C01593=1159.558,276.574,-69.482,-177.157,7.926,148.703
C01594=1159.554,276.823,-69.512,-177.154,7.929,148.703
C01595=1159.549,277.071,-69.540,-177.151,7.932,148.703
C01596=1159.546,277.319,-69.569,-177.148,7.935,148.703
C01597=1159.541,277.567,-69.599,-177.146,7.938,148.703
C01598=1159.537,277.816,-69.627,-177.143,7.941,148.703
C01599=1159.532,278.063,-69.656,-177.140,7.944,148.703
C01600=1159.528,278.312,-69.686,-177.138,7.947,148.703
C01601=1159.523,278.561,-69.715,-177.135,7.950,148.703
C01602=1159.519,278.809,-69.744,-177.133,7.954,148.703
C01603=1159.516,279.057,-69.773,-177.130,7.956,148.703
C01604=1159.512,279.305,-69.802,-177.127,7.959,148.703
C01605=1159.506,279.553,-69.831,-177.124,7.962,148.703
C01606=1159.502,279.801,-69.860,-177.122,7.966,148.703
C01607=1159.498,280.050,-69.890,-177.119,7.969,148.703
C01608=1159.494,280.298,-69.919,-177.116,7.972,148.703
C01609=1159.490,280.546,-69.949,-177.114,7.975,148.703
C01610=1159.486,280.795,-69.978,-177.111,7.978,148.703
C01611=1159.480,281.043,-70.006,-177.109,7.981,148.703
C01612=1159.476,281.291,-70.036,-177.106,7.984,148.703
C01613=1159.472,281.539,-70.065,-177.103,7.987,148.703
C01614=1159.468,281.788,-70.095,-177.101,7.990,148.703
C01615=1159.464,282.036,-70.124,-177.098,7.993,148.703
C01616=1159.460,282.284,-70.154,-177.095,7.996,148.703
C01617=1159.455,282.532,-70.183,-177.093,7.999,148.703
C01618=1159.451,282.781,-70.213,-177.090,8.002,148.703
C01619=1159.446,283.028,-70.242,-177.087,8.005,148.703
C01620=1159.442,283.276,-70.271,-177.085,8.008,148.703
C01621=1159.438,283.525,-70.301,-177.082,8.011,148.703
C01622=1159.434,283.773,-70.330,-177.080,8.014,148.703
C01623=1159.430,284.021,-70.359,-177.077,8.017,148.703
C01624=1159.426,284.270,-70.389,-177.074,8.020,148.703
C01625=1159.421,284.518,-70.419,-177.072,8.023,148.703
C01626=1159.416,284.766,-70.448,-177.069,8.026,148.703
C01627=1159.412,285.015,-70.478,-177.066,8.029,148.703
C01628=1159.408,285.263,-70.507,-177.064,8.032,148.703
C01629=1159.404,285.511,-70.537,-177.061,8.036,148.703
C01630=1159.400,285.759,-70.566,-177.059,8.039,148.703
C01631=1159.396,286.007,-70.596,-177.056,8.042,148.703
C01632=1159.391,286.256,-70.626,-177.053,8.045,148.703
C01633=1159.387,286.504,-70.656,-177.050,8.049,148.703
C01634=1159.383,286.752,-70.685,-177.047,8.052,148.703
C01635=1159.378,287.000,-70.715,-177.045,8.055,148.703
C01636=1159.374,287.249,-70.744,-177.042,8.058,148.703
C01637=1159.370,287.523,-70.778,-177.040,8.061,148.703
C01638=1159.365,287.799,-70.810,-177.036,8.065,148.703
C01639=1159.360,288.074,-70.843,-177.034,8.068,148.703
C01640=1159.355,288.348,-70.877,-177.031,8.072,148.703
C01641=1159.351,288.597,-70.906,-177.028,8.075,148.703
C01642=1159.346,288.845,-70.936,-177.025,8.078,148.704
C01643=1159.342,289.094,-70.966,-177.023,8.081,148.704
C01644=1159.338,289.341,-70.996,-177.020,8.084,148.704
C01645=1159.334,289.589,-71.025,-177.018,8.087,148.704
C01646=1159.329,289.838,-71.055,-177.015,8.090,148.704
C01647=1159.325,290.086,-71.086,-177.012,8.093,148.704
C01648=1159.321,290.334,-71.115,-177.010,8.096,148.704
C01649=1159.316,290.582,-71.146,-177.007,8.099,148.704
C01650=1159.312,290.830,-71.175,-177.004,8.102,148.704
C01651=1159.308,291.078,-71.205,-177.002,8.105,148.704
C01652=1159.304,291.326,-71.235,-176.999,8.108,148.704
C01653=1159.300,291.575,-71.265,-176.997,8.112,148.704
C01654=1159.296,291.823,-71.295,-176.994,8.115,148.704
C01655=1159.291,292.072,-71.326,-176.991,8.118,148.704
C01656=1159.287,292.319,-71.356,-176.989,8.121,148.704
C01657=1159.283,292.567,-71.385,-176.986,8.124,148.704
C01658=1159.278,292.815,-71.416,-176.983,8.128,148.704
C01659=1159.274,293.064,-71.445,-176.981,8.131,148.704
C01660=1159.270,293.311,-71.476,-176.978,8.134,148.704
C01661=1159.265,293.560,-71.506,-176.976,8.137,148.704
C01662=1159.262,293.808,-71.536,-176.973,8.140,148.704
C01663=1159.257,294.057,-71.566,-176.970,8.143,148.704
C01664=1159.253,294.305,-71.596,-176.968,8.146,148.705
C01665=1159.249,294.552,-71.627,-176.965,8.149,148.705
C01666=1159.245,294.801,-71.657,-176.963,8.153,148.705
C01667=1159.241,295.048,-71.687,-176.960,8.155,148.705
C01668=1159.236,295.296,-71.717,-176.957,8.158,148.705
C01669=1159.232,295.545,-71.747,-176.955,8.162,148.705
C01670=1159.228,295.793,-71.778,-176.952,8.165,148.705
C01671=1159.224,296.041,-71.808,-176.949,8.169,148.705
C01672=1159.219,296.289,-71.838,-176.947,8.172,148.705
C01673=1159.215,296.537,-71.868,-176.944,8.175,148.705
C01674=1159.211,296.786,-71.900,-176.942,8.178,148.705
C01675=1159.207,297.034,-71.929,-176.939,8.181,148.705
C01676=1159.202,297.282,-71.960,-176.936,8.184,148.705
C01677=1159.198,297.530,-71.990,-176.934,8.187,148.705
C01678=1159.194,297.778,-72.021,-176.931,8.190,148.705
C01679=1159.190,298.026,-72.052,-176.929,8.193,148.705
C01680=1159.186,298.275,-72.081,-176.926,8.197,148.706
C01681=1159.181,298.523,-72.112,-176.924,8.200,148.706
C01682=1159.177,298.770,-72.142,-176.921,8.204,148.706
C01683=1159.173,299.019,-72.173,-176.918,8.207,148.706
C01684=1159.169,299.267,-72.204,-176.915,8.210,148.706
C01685=1159.165,299.514,-72.234,-176.913,8.213,148.706
C01686=1159.160,299.763,-72.264,-176.910,8.216,148.706
C01687=1159.157,300.011,-72.295,-176.908,8.219,148.706
C01688=1159.152,300.259,-72.326,-176.905,8.222,148.706
C01689=1159.147,300.507,-72.356,-176.903,8.225,148.706
C01690=1159.143,300.755,-72.387,-176.900,8.228,148.706
C01691=1159.139,301.004,-72.418,-176.897,8.233,148.706
C01692=1159.135,301.252,-72.448,-176.894,8.235,148.706
C01693=1159.131,301.499,-72.479,-176.892,8.239,148.707
C01694=1159.127,301.748,-72.510,-176.889,8.242,148.706
C01695=1159.122,301.996,-72.541,-176.887,8.245,148.707
C01696=1159.118,302.244,-72.571,-176.884,8.248,148.707
C01697=1159.114,302.492,-72.602,-176.882,8.251,148.707
C01698=1159.110,302.740,-72.633,-176.879,8.254,148.707
C01699=1159.105,302.988,-72.663,-176.877,8.258,148.707
C01700=1159.101,303.236,-72.694,-176.874,8.261,148.707
C01701=1159.097,303.484,-72.725,-176.871,8.265,148.707
C01702=1159.093,303.732,-72.756,-176.869,8.268,148.707
C01703=1159.088,303.980,-72.787,-176.866,8.271,148.707
C01704=1159.084,304.228,-72.818,-176.863,8.274,148.707
C01705=1159.080,304.476,-72.849,-176.861,8.277,148.707
C01706=1159.076,304.725,-72.879,-176.858,8.280,148.707
C01707=1159.072,304.973,-72.910,-176.856,8.284,148.708
C01708=1159.068,305.220,-72.942,-176.853,8.287,148.708
C01709=1159.064,305.469,-72.973,-176.850,8.290,148.708
C01710=1159.059,305.716,-73.003,-176.848,8.294,148.708
C01711=1159.054,305.964,-73.034,-176.845,8.297,148.708
C01712=1159.051,306.213,-73.065,-176.843,8.300,148.708
C01713=1159.047,306.460,-73.096,-176.840,8.303,148.708
C01714=1159.043,306.709,-73.127,-176.837,8.307,148.708
C01715=1159.038,306.957,-73.158,-176.835,8.310,148.708
C01716=1159.034,307.204,-73.190,-176.832,8.313,148.709
C01717=1159.030,307.453,-73.221,-176.830,8.316,148.709
C01718=1159.025,307.701,-73.252,-176.827,8.319,148.709
C01719=1159.021,307.949,-73.283,-176.825,8.323,148.709
C01720=1159.017,308.197,-73.314,-176.822,8.326,148.709
C01721=1159.013,308.445,-73.345,-176.819,8.330,148.709
C01722=1159.009,308.693,-73.377,-176.817,8.333,148.709
C01723=1159.004,308.941,-73.407,-176.814,8.336,148.709
C01724=1159.000,309.189,-73.439,-176.812,8.339,148.709
C01725=1158.996,309.436,-73.470,-176.809,8.342,148.709
C01726=1158.992,309.685,-73.501,-176.807,8.346,148.710
C01727=1158.988,309.932,-73.532,-176.804,8.349,148.710
C01728=1158.984,310.181,-73.563,-176.801,8.353,148.710
C01729=1158.980,310.428,-73.595,-176.799,8.356,148.710
C01730=1158.976,310.677,-73.626,-176.796,8.359,148.710
C01731=1158.971,310.924,-73.657,-176.794,8.362,148.710
C01732=1158.967,311.173,-73.689,-176.791,8.365,148.710
C01733=1158.962,311.421,-73.721,-176.788,8.369,148.710
C01734=1158.958,311.669,-73.752,-176.786,8.373,148.711
C01735=1158.954,311.917,-73.783,-176.783,8.375,148.711
C01736=1158.950,312.165,-73.815,-176.781,8.379,148.711
C01737=1158.946,312.413,-73.846,-176.779,8.382,148.711
C01738=1158.942,312.661,-73.878,-176.776,8.385,148.711
C01739=1158.937,312.909,-73.908,-176.773,8.389,148.711
C01740=1158.934,313.157,-73.940,-176.770,8.392,148.711
C01741=1158.929,313.433,-73.975,-176.768,8.395,148.711
C01742=1158.924,313.711,-74.011,-176.765,8.399,148.712
C01743=1158.919,313.988,-74.046,-176.762,8.403,148.712
C01744=1158.915,314.266,-74.081,-176.759,8.407,148.712
C01745=1158.911,314.514,-74.113,-176.757,8.411,148.712
C01746=1158.907,314.761,-74.145,-176.754,8.414,148.712
C01747=1158.903,315.010,-74.176,-176.752,8.417,148.712
C01748=1158.898,315.258,-74.208,-176.749,8.420,148.712
C01749=1158.894,315.506,-74.240,-176.746,8.424,148.712
C01750=1158.890,315.753,-74.271,-176.744,8.427,148.713
C01751=1158.886,316.002,-74.302,-176.741,8.431,148.713
C01752=1158.882,316.250,-74.334,-176.739,8.433,148.713
C01753=1158.877,316.497,-74.366,-176.736,8.437,148.713
C01754=1158.873,316.745,-74.398,-176.733,8.441,148.713
C01755=1158.870,316.993,-74.430,-176.731,8.444,148.713
C01756=1158.865,317.241,-74.461,-176.728,8.447,148.713
C01757=1158.861,317.489,-74.494,-176.726,8.450,148.714
C01758=1158.857,317.738,-74.525,-176.723,8.453,148.713
C01759=1158.853,317.985,-74.556,-176.720,8.457,148.714
C01760=1158.849,318.233,-74.588,-176.718,8.461,148.714
C01761=1158.844,318.481,-74.620,-176.715,8.464,148.714
C01762=1158.840,318.729,-74.652,-176.713,8.467,148.714
C01763=1158.836,318.977,-74.684,-176.711,8.470,148.714
C01764=1158.833,319.225,-74.716,-176.708,8.474,148.715
C01765=1158.828,319.473,-74.748,-176.705,8.477,148.715
C01766=1158.824,319.721,-74.780,-176.703,8.481,148.715
C01767=1158.820,319.969,-74.812,-176.700,8.484,148.715
C01768=1158.815,320.216,-74.844,-176.698,8.488,148.715
C01769=1158.811,320.464,-74.875,-176.695,8.491,148.715
C01770=1158.808,320.712,-74.907,-176.693,8.494,148.715
C01771=1158.803,320.960,-74.939,-176.690,8.498,148.715
C01772=1158.799,321.208,-74.971,-176.687,8.501,148.715
C01773=1158.795,321.456,-75.004,-176.685,8.505,148.716
C01774=1158.791,321.704,-75.036,-176.682,8.508,148.716
C01775=1158.787,321.951,-75.068,-176.680,8.511,148.716
C01776=1158.782,322.200,-75.100,-176.678,8.514,148.716
C01777=1158.779,322.448,-75.132,-176.674,8.518,148.716
C01778=1158.774,322.696,-75.164,-176.672,8.522,148.717
C01779=1158.770,322.943,-75.196,-176.670,8.525,148.717
C01780=1158.766,323.191,-75.229,-176.667,8.528,148.717
C01781=1158.762,323.439,-75.261,-176.664,8.532,148.717
C01782=1158.758,323.687,-75.293,-176.662,8.535,148.717
C01783=1158.754,323.935,-75.325,-176.659,8.538,148.717
C01784=1158.750,324.182,-75.357,-176.657,8.542,148.718
C01785=1158.746,324.430,-75.390,-176.654,8.546,148.718
C01786=1158.742,324.679,-75.422,-176.652,8.549,148.718
C01787=1158.737,324.927,-75.454,-176.649,8.552,148.718
C01788=1158.734,325.174,-75.487,-176.647,8.555,148.718
C01789=1158.729,325.422,-75.519,-176.644,8.559,148.718
C01790=1158.725,325.670,-75.551,-176.641,8.562,148.718
C01791=1158.721,325.918,-75.584,-176.639,8.566,148.719
C01792=1158.717,326.166,-75.616,-176.637,8.569,148.719
C01793=1158.713,326.413,-75.649,-176.634,8.573,148.719
C01794=1158.708,326.661,-75.681,-176.632,8.576,148.719
C01795=1158.704,326.909,-75.713,-176.629,8.580,148.719
C01796=1158.700,327.157,-75.746,-176.626,8.583,148.719
C01797=1158.696,327.405,-75.778,-176.624,8.587,148.720
C01798=1158.692,327.653,-75.811,-176.621,8.590,148.720
C01799=1158.688,327.901,-75.843,-176.619,8.593,148.720
C01800=1158.685,328.148,-75.876,-176.616,8.597,148.720
C01801=1158.680,328.396,-75.908,-176.614,8.601,148.720
C01802=1158.675,328.644,-75.941,-176.611,8.604,148.720
C01803=1158.672,328.892,-75.973,-176.609,8.607,148.721
C01804=1158.668,329.140,-76.006,-176.606,8.611,148.721
C01805=1158.663,329.388,-76.039,-176.604,8.614,148.721
C01806=1158.660,329.635,-76.071,-176.601,8.618,148.721
C01807=1158.655,329.884,-76.104,-176.598,8.622,148.722
C01808=1158.651,330.131,-76.137,-176.596,8.625,148.722
C01809=1158.647,330.379,-76.170,-176.593,8.628,148.722
C01810=1158.643,330.627,-76.202,-176.591,8.631,148.722
C01811=1158.639,330.874,-76.234,-176.588,8.635,148.722
C01812=1158.634,331.123,-76.267,-176.586,8.639,148.722
C01813=1158.631,331.370,-76.299,-176.583,8.642,148.723
C01814=1158.627,331.618,-76.333,-176.581,8.646,148.723
C01815=1158.622,331.866,-76.365,-176.578,8.649,148.723
C01816=1158.618,332.114,-76.398,-176.576,8.653,148.723
C01817=1158.614,332.362,-76.431,-176.573,8.657,148.723
C01818=1158.610,332.609,-76.464,-176.570,8.660,148.723
C01819=1158.606,332.857,-76.496,-176.568,8.663,148.724
C01820=1158.602,333.105,-76.530,-176.566,8.666,148.724
C01821=1158.598,333.353,-76.563,-176.563,8.670,148.724
C01822=1158.594,333.600,-76.596,-176.561,8.674,148.724
C01823=1158.590,333.849,-76.628,-176.558,8.677,148.725
C01824=1158.586,334.096,-76.661,-176.555,8.681,148.725
C01825=1158.582,334.344,-76.694,-176.553,8.684,148.725
C01826=1158.578,334.592,-76.727,-176.551,8.688,148.725
